fb_sdoread_6041(sNetId:= fb_netid, nSlaveAddr:=fb_nslaveaddr , nSubIndex:=0 , nIndex:=16#6041 , pDstBuf:=ADR(statusword) , cbBufLen:=2 , bExecute:=sdo_read , tTimeout:= , bBusy=> , bError=> , nErrId=> );
fb_sdoread_6060(sNetId:= fb_netid, nSlaveAddr:= fb_nslaveaddr, nSubIndex:=0 , nIndex:=16#6060 , pDstBuf:=ADR(mode_display) , cbBufLen:=1 , bExecute:=sdo_read , tTimeout:= , bBusy=> , bError=> , nErrId=> );
//fb_sdowrite_6060(sNetId:= fb_netid, nSlaveAddr:=fb_nslaveaddr , nSubIndex:=0 , nIndex:= 16#6060, pSrcBuf:=ADR(mode) , cbBufLen:=1 , bExecute:= mode<>mode_display AND sdo_read, tTimeout:= , bBusy=> , bError=> , nErrId=> );
fb_sdoread_607C(sNetId:= fb_netid, nSlaveAddr:=fb_nslaveaddr , nSubIndex:=0 , nIndex:=16#607C , pDstBuf:= ADR(home_offset_display), cbBufLen:=4 , bExecute:=sdo_read , tTimeout:= , bBusy=> , bError=> , nErrId=> );
fb_sdowrite_607C(sNetId:=fb_netid , nSlaveAddr:=fb_nslaveaddr , nSubIndex:=0 , nIndex:=16#607C , pSrcBuf:=ADR(home_offset) , cbBufLen:=4 ,	bExecute:=home_offset<>home_offset_display AND sdo_read , tTimeout:= , bBusy=> , bError=> , nErrId=> );
fb_sdoread_6098(sNetId:=fb_netid , nSlaveAddr:=fb_nslaveaddr , nSubIndex:=0 , nIndex:=16#6098 , pDstBuf:=ADR(home_method_display) , cbBufLen:=1 , bExecute:=sdo_read , tTimeout:= , bBusy=> , bError=> , nErrId=> );
fb_sdowrite_6098(sNetId:=fb_netid , nSlaveAddr:=fb_nslaveaddr , nSubIndex:=0 , nIndex:=16#6098 , pSrcBuf:=ADR(home_method) , cbBufLen:=1 , bExecute:=home_method<>home_method_display AND sdo_read , tTimeout:= , bBusy=> , bError=> , nErrId=> );
fb_sdoread_6099_01(sNetId:=fb_netid , nSlaveAddr:=fb_nslaveaddr , nSubIndex:=1 , nIndex:=16#6099, pDstBuf:=ADR(home_highspeed_display) , cbBufLen:=4 , bExecute:=sdo_read , tTimeout:= , bBusy=> , bError=> , nErrId=> );
fb_sdowrite_6099_01(sNetId:=fb_netid , nSlaveAddr:=fb_nslaveaddr , nSubIndex:=1 , nIndex:=16#6099 , pSrcBuf:=ADR(home_highspeed) , cbBufLen:=4 , bExecute:=home_highspeed<>home_highspeed_display AND sdo_read , tTimeout:= , bBusy=> , bError=> , nErrId=> );
fb_sdoread_6099_02(sNetId:=fb_netid , nSlaveAddr:=fb_nslaveaddr , nSubIndex:=2 , nIndex:=16#6099, pDstBuf:= ADR(home_lowspeed_display), cbBufLen:= 4, bExecute:=sdo_read , tTimeout:= , bBusy=> , bError=> , nErrId=> );
fb_sdowrite_6099_02(sNetId:=fb_netid , nSlaveAddr:=fb_nslaveaddr , nSubIndex:=2 , nIndex:=16#6099 , pSrcBuf:=ADR(home_lowspeed) , cbBufLen:=4 , bExecute:=home_lowspeed<>home_lowspeed_display AND sdo_read , tTimeout:= , bBusy=> , bError=> , nErrId=> );
fb_sdoread_6091_01(sNetId:=fb_netid , nSlaveAddr:=fb_nslaveaddr , nSubIndex:=1 , nIndex:=16#6091 , pDstBuf:= ADR(motor), cbBufLen:= 4, bExecute:=sdo_read , tTimeout:= , bBusy=> , bError=> , nErrId=> );
fb_sdoread_6091_02(sNetId:=fb_netid , nSlaveAddr:=fb_nslaveaddr , nSubIndex:=2 , nIndex:=16#6091 , pDstBuf:=ADR(shaft), cbBufLen:=4 , bExecute:=sdo_read , tTimeout:= , bBusy=> , bError=> , nErrId=> );
//fb_sdoread_6064(sNetId:=fb_netid , nSlaveAddr:=fb_nslaveaddr , nSubIndex:=2 , nIndex:=16#6099 , pSrcBuf:=ADR(home_lowspeed) , cbBufLen:=4 , bExecute:=home_lowspeed<>home_lowspeed_display AND sdo_read , tTimeout:= , bBusy=> , bError=> , nErrId=> );

IF iMode = 3 OR iMode =1 //雷赛伺服
THEN 
	mcsetposition(
		Axis:= axis_name, 
		Execute:= (statusword.10=TRUE AND  statusword.12=TRUE AND statusword.13=FALSE AND home_start), 
		Position:= 0, 
		Mode:= , 
		Options:= , 
		Done=> , 
		Busy=> , 
		Error=> , 
		ErrorID=> );
END_IF

IF home_exe THEN
home_start:=TRUE;
home_done := FALSE;//增加
//ELSE home_error:=TRUE; error_id:=8001; home_start:=FALSE;
END_IF

IF home_start (*AND FALSE*) THEN
	CASE home_step OF
		0://复位关闭
		exe_reset:=FALSE;	
		IF NOT(home_error) THEN
			home_step:=3;
			mcsetposition(
				Axis:= axis_name, 
				Execute:= FALSE);
		END_IF
		1://检测是否是三菱驱动器
		IF 	iMode = 1
		THEN 
			mcsetposition(
			Axis:= axis_name, 
			Execute:= TRUE, 
			Position:= 0, 
			Mode:= , 
			Options:= , 
			Done=> , 
			Busy=> , 
			Error=> , 
			ErrorID=> ); 
			IF mcsetposition.Done
			THEN
				mcsetposition(
					Axis:= axis_name, 
					Execute:= FALSE);
				home_step := 3;
			END_IF			
		ELSE
			home_step := 3; 
		END_IF
		
		3://将模式切为回原点模式6
		mode:=6;
		home_done := FALSE;
		ton2.IN:=TRUE;
		IF ton2.Q THEN
			ton2.IN:=FALSE;
			home_step:=5;
		END_IF
		5://将控制字改为F，上使能
        IF NOT home_error THEN
			controlword:=15;
			home_step:=10;
			ton2.IN:=FALSE;
		ELSE
			home_error:=TRUE;
			error_id:=8002;
			home_step:=0;
		END_IF
		10://复位
		exe_reset:=TRUE;
		ton2.IN:=TRUE;
		IF ton2.Q THEN 
			ton2.IN:=FALSE;
			home_step:=15;
		END_IF
		15://复位完成，控制字改为F
		IF reset_done AND statusword.1 THEN
			exe_reset:=FALSE;
			home_step:=25;
		ELSE
			home_error:=TRUE;
			error_id:=8003;
			home_step:=0;
		END_IF
		
		25://确认模式切换为6,与设定值相同
		IF mode=mode_display AND home_offset=home_offset_display AND home_method=home_method_display AND home_highspeed=home_highspeed_display AND home_lowspeed=home_lowspeed_display 
        AND (mode_display<>0) AND (home_method_display<>0) AND (home_highspeed_display<>0) AND (home_lowspeed_display<>0) AND (numerator<>0) AND (denominator<>0) THEN 
			home_step:=26;
			_tonDelay1(in:=FALSE);
			_tonDelay2(in:=FALSE);
		ELSE
			home_error:=TRUE;
			error_id:=8004;
			home_step:=0;
		END_IF
		
		26:
			controlword:=31;
			_tonDelay1(in:=TRUE,PT:=T#2S);
			IF _tonDelay1.Q THEN
				_tonDelay1(in:=FALSE);
				home_step:=30;
			END_IF		
		30://将控制字切为1F，启动回原点功能
		IF statusword.10 AND  statusword.12 AND NOT statusword.13 THEN
			home_step:=40;
		(*ELSIF statusword.13 THEN
			home_error:=TRUE;
			error_id:=8005;
			home_step:=0;	*)		
		ELSE
			_tonDelay2(IN:=TRUE,pt:=tTimeOutSet);
		END_IF
		
		(*_tonDelay1(in:=(statusword.10=TRUE) AND  statusword.12=TRUE AND statusword.13=FALSE,pt:=T#200MS);//回原点已经完成
		_tonDelay2(in:=( statusword.10=FALSE AND  statusword.12=FALSE AND statusword.13=TRUE ) OR ( statusword.10=FALSE AND  statusword.12=TRUE AND statusword.13=FALSE ) OR 
                       ( statusword.10=TRUE AND  statusword.12=FALSE AND statusword.13=FALSE ) OR ( statusword.10=TRUE AND  statusword.12=FALSE AND statusword.13=TRUE ) OR 
					   ( statusword.12=TRUE AND statusword.13=TRUE )	,pt:=T#10S);//会员店内失败
		IF _tonDelay1.Q  THEN//检测状态字回原点完成
			_tonDelay1(IN:=FALSE);
			home_step:=40;
		END_IF*)
		IF _tonDelay2.Q THEN
			_tonDelay2(IN:=FALSE);
			home_error:=TRUE;
			error_id:=8005;
			home_step:=0;
		END_IF
		40://复位
		//exe_reset:=TRUE;
		_tonDelay2(IN:=FALSE);
		ton2.IN:=(TRUE);
		IF ton2.Q THEN
			ton2.IN:=(FALSE);
			_tonDelay(IN:=FALSE);
			home_step:=41;
		END_IF
		41://增加断使能功能
		controlword:=0;
		_tonDelay(IN:=NOT statusword.1 , PT:=T#100MS , Q=> , ET=> );
		IF _tonDelay.Q THEN
			_tonDelay(IN:=FALSE);
			home_step:=45;
		END_IF

		45://将模式切换为位置模式8
//		IF reset_done THEN			
//			exe_reset:=FALSE;
//			_tonDelay(IN:=FALSE);
			home_step:=46;
//		ELSE
//			home_error:=TRUE;
//			error_id:=8006;
//			home_step:=0;
//		END_IF
		46://增加上使能功能
		//controlword:=15;
		_tonDelay(IN:=TRUE , PT:=T#1S , Q=> , ET=> );
		IF _tonDelay.Q THEN
			_tonDelay(IN:=FALSE);
			home_step:=50;
		END_IF		
		50:
		_iCount := _iCount + 1 ;
		mode:=8;
		home_done:=TRUE;
		exe_reset:=FALSE;
		home_start:=FALSE;
		home_step:=0;
	END_CASE
END_IF


(*IF NOT(home_exe)THEN
	home_step:=0;
	home_error:=FALSE;
	home_done:=FALSE;
	home_start:=FALSE;
	error_id:=0;
END_IF*)

IF home_error THEN
	home_step:=0;
	//
	home_done:=FALSE;
	home_start:=FALSE;
	exe_reset:=TRUE;
	IF reset_done THEN
		error_id:=0;
		mode:=8;
		home_error:=FALSE;
		exe_reset:=FALSE;
	END_IF
END_IF

END_FUNCTION_BLOCK

// ---- POUs/003_FB/17_HMIFB/FB_Proface.TcPOU
FUNCTION_BLOCK FB_Proface
VAR_INPUT
	xEStop								: BOOL;					//急停
	xSafety								: BOOL;					//安全防护
	xManualMode							: BOOL;					//手动模式
	xAutoMode							: BOOL;					//自动模式
	xAlarm								: BOOL;					//报警中
	xTip								: BOOL;					//提示中
	xInit								: BOOL;					//初始化
	xIniting							: BOOL;					//初始化中
	xInitDone							: BOOL;					//初始化完成
	xDummyChecking						: BOOL;					//点检中
	xDummyCheckDone						: BOOL;					//点检完成
	xEmptying							: BOOL;					//清料中
	xEmptyDone							: BOOL;					//清料完成
	xStartHmi							: BOOL;					//启动HMI
	xStopHmi							: BOOL;					//停止HMI
	xResetHmi							: BOOL;					//复位HMI
	xPauseHmi							: BOOL;					//暂停HMI
	xInitHmi							: BOOL;					//初始化HMI
	xInitConfirmHmi						:BOOL;					//测试使用
	xManualModeHmi						: BOOL;					//手动HMI
	xAutoModeHmi						: BOOL;					//自动HMI
	xUnlockHmi							: BOOL;					//解锁HMI
	xDummyCheckHmi						: BOOL;					//点检HMI
	xEmptyHmi							: BOOL;					//清料HMI
	xWindowColseHmi						: BOOL;					//窗口关闭HMI
	                      		
	nCurrentPageIndex					: UINT:=0;				//当前画面索引
	nJumpToPageIndex					: UINT:=1;				//跳转到画面索引
	                      		
	nWindowControlIndex					: UINT:=0;				//窗口控制索引
	nWindowNumberIndex					: UINT:=1;				//窗口编号索引
	nWindowLocationIndexX				: UINT:=2;				//窗口位置索引X坐标
	nWindowLocationIndexY				: UINT:=3;				//窗口位置索引Y坐标
	                      		
	nWindowLocationX					: UINT:=300;			//窗口位置X坐标
	nWindowLocationY					: UINT:=80;		    //窗口位置Y坐标
	                      		
	nInitConfirmWindow					: UINT:=1;				//初始化确认窗口编号
	nInitAlarmWindow					: UINT:=2;				//初始化有报警窗口编号
	nInitingAlarmWindow					: UINT:=3;				//初始化中有报警窗口编号
	nInitingWindow						: UINT:=4;				//初始化中窗口编号
	nInitDoneWindow						: UINT:=5;				//初始化完成窗口编号
	nInitFailWindow						: UINT:=6;				//初始化失败窗口编号
	
	nDummyCheckConfirmWindow			: UINT:=5;				//点检确认窗口编号
	nDummyCheckDoneWindow				: UINT:=6;				//点检完成窗口编号
	nDummyCheckFailWindow				: UINT:=7;				//点检失败窗口编号
	
	nEmptyConfirmWindow					: UINT:=10;				//清料确认窗口编号
	nEmptyDoneWindow					: UINT:=11;				//清料完成窗口编号
	
	nTipWindow							: UINT:=31;				//提示窗口编号
	nButtonWindow						: UINT:=121;			//调试窗口编号
END_VAR

VAR_OUTPUT
END_VAR

VAR
	
	xStartLight							: BOOL;					//启动灯
	xStopLight							: BOOL;					//停止灯
	xResetLight							: BOOL;					//复位灯
	xPauseLight							: BOOL;					//暂停灯
	xInitLight							: BOOL;					//初始化灯
	
END_VAR

VAR
	
	wSystem								: ARRAY[0..20] OF WORD;	//系统区
	wWindow								: ARRAY[0..20] OF WORD;	//窗口控制区
	                  				
	ftTip								: F_TRIG;				//提示中下降沿
	rtInit								: R_TRIG;				//初始化上升沿
	ftIniting							: F_TRIG;				//初始化中下降沿
	rtDummyCheck						: R_TRIG;				//点检上升沿
	ftDummyChecking						: F_TRIG;				//点检中下降沿
	rtEmptyConfirm						: R_TRIG;				//清料确认上升沿
	rtEmptyDone							: R_TRIG;				//清料完成上升沿
	
END_VAR

ACT_Init();
ACT_DummyCheck();
ACT_Empty();
ACT_Control();

ACTION ACT_Control:
ftTip(CLK:=xTip, Q=>);
IF xWindowColseHMI		//窗口关闭
	OR ftTip.Q			//提示下降沿自动关闭窗口
THEN
	wWindow[nWindowNumberIndex]:=0;
END_IF

//IF xTip THEN
//	wWindow[nWindowNumberIndex]:=nTipWindow;
//END_IF

wWindow[nWindowControlIndex].0:=wWindow[nWindowNumberIndex]<>0;

wWindow[nWindowLocationIndexX]:=nWindowLocationX;
wWindow[nWindowLocationIndexY]:=nWindowLocationY;
END_ACTION

ACTION ACT_DummyCheck:
rtDummyCheck(CLK:=xDummyCheckHmi, Q=>);
ftDummyChecking(CLK:=xDummyChecking, Q=>);
IF rtDummyCheck.Q	//点检确认窗口显示
	AND xEStop
	AND xSafety
	AND xManualMode
	AND xInitDone
	AND NOT xAlarm
THEN
	wWindow[nWindowNumberIndex]:=nDummyCheckConfirmWindow;
END_IF
IF ftDummyChecking.Q THEN
	IF xDummyCheckDone THEN		//点检完成窗口显示
		wWindow[nWindowNumberIndex]:=nDummyCheckDoneWindow;
	ELSE	//点检失败窗口显示
		wWindow[nWindowNumberIndex]:=nDummyCheckFailWindow;
	END_IF
END_IF
END_ACTION

ACTION ACT_Empty:
rtEmptyConfirm(CLK:=xEmptyHmi, Q=>);
rtEmptyDone(CLK:=xEmptyDone, Q=>);
IF rtEmptyConfirm.Q		//清料确认窗口显示
	AND fbMachine[1].xEStop
	AND fbMachine[1].xSafety
	AND fbMachine[1].xAutoMode
	AND fbMachine[1].xInitDone
	AND NOT fbMachine[1].xAlarm
THEN
	wWindow[nWindowNumberIndex]:=nEmptyConfirmWindow;
END_IF

IF rtEmptyDone.Q THEN	//清料完成窗口显示
	wWindow[nWindowNumberIndex]:=nEmptyDoneWindow;
END_IF
END_ACTION

ACTION ACT_Init:
rtInit(CLK:=xInit, Q=>);
ftIniting(CLK:=xIniting, Q=>);

IF rtInit.Q
THEN
	wSystem[0]:=10;
END_IF

IF rtInit.Q					//初始化确认窗口显示
	AND xEStop
	AND xSafety
	AND xManualMode
	AND NOT xAlarm
	AND NOT xIniting
THEN
	wWindow[nWindowNumberIndex]:=nInitConfirmWindow;
END_IF

IF rtInit.Q					//初始化有报警
	AND xAlarm
THEN
	wWindow[nWindowNumberIndex]:=nInitAlarmWindow;
END_IF

IF xIniting					//初始化中有报警
	AND xAlarm
THEN
	wWindow[nWindowNumberIndex]:=nInitingAlarmWindow;
END_IF

IF xIniting THEN			//初始化中窗口显示
	wWindow[nWindowNumberIndex]:=nInitingWindow;
END_IF

IF ftIniting.Q THEN		
	IF xInitDone THEN		//初始化完成窗口显示
		wWindow[nWindowNumberIndex]:=nInitDoneWindow;
	ELSE					//初始化失败窗口显示
		wWindow[nWindowNumberIndex]:=nInitFailWindow;
	END_IF
END_IF

IF xWindowColseHMI
THEN
	wWindow[nWindowNumberIndex]:=0;
	wWindow[nWindowControlIndex]:=0;
END_IF
END_ACTION

END_FUNCTION_BLOCK

// ---- POUs/003_FB/14_MachineFB/FB_Machine.TcPOU
FUNCTION_BLOCK  FB_Machine
VAR_INPUT
	xEStop						: BOOL;					//急停(运行时常ON)
	xKey						: BOOL;					//钥匙开关
	xDoorClosed					: BOOL;					//所有安全门关好
	xSafety						: BOOL;					//安全防护中
	xAirOn						: BOOL;					//气压正常
	xAlarm						: BOOL;					//报警中
	xManualTip					: BOOL;					//手动提示中
	xAutoTip					: BOOL;					//自动提示中
	xTip						: BOOL;					//提示中
	
	xStart						: BOOL;					//启动按钮
	xStop						: BOOL;					//停止按钮
	xReset						: BOOL;					//复位按钮
	xPause						: BOOL;					//暂停按钮
	xInit						: BOOL;					//初始化按钮
	xManualMode					: BOOL;					//手动模式
	xAutoMode					: BOOL;					//自动模式

	
	xInitConfirm				: BOOL;					//初始化确认
	xInitDone					: BOOL;					//初始化完成
	tInitTimeout				: TIME:=T#3M;			//初始化超时延时
	
	xDummyMode					: BOOL;					//点检模式，点检使能
	xStationDummyDone			: BOOL;					//工站点检完成
	xDummyDone					: BOOL;					//点检完成
	xDummyDoneConfirm			: BOOL;					//点检完成确认
	
	xSampling					: BOOL;					//取样中
	uiSampleCount				: UINT;					//取样数量统计
	xSampleDone					: BOOL;					//取样完成
	xEmptyHmi					: BOOL;					//清料HMI
	xEmptyConfirmHmi			: BOOL;					//清料确认HMI
	xEmptyDone					: BOOL;					//清料完成
	xOrderFinished				: BOOL;					//订单完成
	xOrderChanged				: BOOL;					//订单切换
	
	xTryRun						: BOOL;					//空跑试运行
	xCycleEnable      	 		: BOOL;          		//设备CT计时
	xDataEmpty					: BOOL;					//数据清空
	tDataEmpty					: TIME;					//数据清空延时，默认为0
	xCarrierDataClear			: BOOL;					//载座数据清空
	tCarrierDataClear			: TIME;					//载座数据清空延时，默认为0
	
	xInitConfirmDialog			: BOOL;					//初始化确认对话框
	
	dwStatus					:ARRAY[1..4] OF DWORD;	//状态，bit.0急停中.1钥匙关闭.2气压低.3手动模式.4自动模式.5未准备好.6准备就绪.7运行中.8停止中.9报警中.10暂停中.11初始化中.12清料中.13清料完成.14取样中.15取样完成.16订单完成.17点检屏蔽中.18要求点检.其它可自定义	
 
	dwMessage					:ARRAY[1..5] OF DWORD;	//提示信息
	dwAlarm						:ARRAY[1..5] OF DWORD;	//报警信息	
	
	xDummyDisabled				: REFERENCE TO BOOL;	//点检屏
	//rCycleTime				: REAL;					//生产周期，单位s
	//生产信息相关变量
	xClearCountData 			: BOOL ; //清除产量数据
	udiGoods					: UDINT;				//当前良品数量
	udiBads						: UDINT;				//当前不良数量
	udiTotal					:  UDINT;				//当前总数量
	rYield						:  REAL;				//当前良品率
	rReject						:  REAL;				//当前不良率
END_VAR

VAR_OUTPUT
	xEStopped					: BOOL;					//急停状态
	xRunning					: BOOL;					//自动中
	xStopped					: BOOL;					//停止状态
	xPaused						: BOOL;					//暂停状态
	xIniting					: BOOL;					//初始化中
	xEmptying					: BOOL;					//清料中
	
	xAutoModeTip				: BOOL;					//自动模式上升沿提示
	
	xInitTimeout				: BOOL;					//初始化超时
	xReInit						: BOOL;					//整机重新初始化，用于复位各工站初始化完成
	
	xInitDoneDialog				: BOOL;					//初始化完成对话框
	xInitFailedDialog			: BOOL;					//初始化失败对话框
	
	xEmptyConfirmDialog			: BOOL;					//清料确认对话框
	xEmptyDoneDialog			: BOOL;					//清料完成对话框
	
	xShowAlarm					: BOOL;					//报警信息显示
	xShowTip					: BOOL;					//提示信息显示
	
	xStartLight					: BOOL;					//启动按钮灯
	xStopLight					: BOOL;					//停止按钮灯
	xResetLight					: BOOL;					//复位按钮灯
	xPauseLight					: BOOL;					//暂停按钮灯
	xInitLight					: BOOL;					//初始化按钮灯
	
	xLampGreen					: BOOL;					//三色灯-绿
	xLampYellow					: BOOL;					//三色灯-黄
	xLampRed					: BOOL;					//三色灯-红
	xLampBuzzer					: BOOL;					//三色灯-蜂鸣器	
	
	diLastCycleTime				:DINT;					//基础时间是100ms
	diCycleTime        			: DINT;					//基础时间是100ms

END_VAR

VAR
	{attribute 'hide'}
	rtRunning					: R_TRIG;				//自动中上升沿
	{attribute 'hide'}
	rtEmptyDone					: R_TRIG;				//清料完成上升沿
	{attribute 'hide'}
	tonDataEmpty				: TON;					//数据清零延时
	rtDataEmpty					: R_TRIG;				//数据清空上升沿
	{attribute 'hide'}
	tonCarrierDataClear			: TON;					//载座数据清空延时
	rtCarrierDataClear			: R_TRIG;				//载座数据清空上升沿
	{attribute 'hide'}
	xDummyWarnTime				: BOOL;					//点检提醒时间
	{attribute 'hide'}
	rtDummyWarnTime				: R_TRIG;				//点检提醒时间上升沿
	{attribute 'hide'}
	xDummyAlarmTime				: BOOL;					//点检报警时间
	{attribute 'hide'}
	rtDummyAlarmTime			: R_TRIG;				//点检报警时间上升沿
	{attribute 'hide'}
	rtDummyDoneConfirm			: R_TRIG;				//点检完成确认上升沿
	{attribute 'hide'}
	xDummyDoneCache				: BOOL;					//点检完成缓存
	{attribute 'hide'}
	xDummyComplete				: BOOL;					//点检完成状态
	{attribute 'hide'}
	xDummyRequirement			: BOOL;					//要求点检提醒
	{attribute 'hide'}
	rtInit						: R_TRIG;				//初始化上升沿
	{attribute 'hide'}
	rtInitConfirm				: R_TRIG;				//初始化确认上升沿
	{attribute 'hide'}
	ftIniting					: F_TRIG;				//初始化下降沿
	{attribute 'hide'}
	rtEmptyHmi					: R_TRIG;				//清料HMI上升沿
	{attribute 'hide'}
	ftEmptying					: F_TRIG;				//清料中下降沿
	{attribute 'hide'}
	xInitAble					: BOOL;					//初始化条件
	{attribute 'hide'}
	xRunAble					: BOOL;					//运行条件
	{attribute 'hide'}
	tonInitTimeout				: TON;					//初始化超时
	{attribute 'hide'}
	tonLampBuzzer				: TON;					//蜂鸣器关闭延时
	{attribute 'hide'}
	rtCycleFlag					: R_TRIG;				//循环标志上升沿
	{attribute 'hide'}
	lrCycleTimer				: LREAL;				//计时器，单位100ns，除于10000后单位ms
	{attribute 'hide'}
	tonHydraGoodsOut			: TON;					//Hydra良品输出信号延时
	{attribute 'hide'}
	tonHydraGoodsInterval		: TON;					//Hydra良品输出信号间隔
	{attribute 'hide'}
	tonHydraBadsOut				: TON;					//Hydra不良输出信号延时
	{attribute 'hide'}
	tonHydraBadsInterval		: TON;					//Hydra不良输出信号间隔
	
	rtAutoMode					: R_TRIG;				//自动模式上升沿
	rMachineStart       		: R_TRIG;
	i : INT ;

END_VAR

ACT_General();
ACT_Init();
ACT_Empty();
ACT_Start();
ACT_Pause();
ACT_Stop();
ACT_Reset();
ACT_Lamp();
ACT_Data();
ACT_CycleTime();

ACTION ACT_CycleTime:
//	初始化时同时初始化工站周期计时
IF xIniting THEN
	xCycleEnable:=FALSE;
END_IF

//工站完成触发信号
rMachineStart(CLK:= xCycleEnable);
IF rMachineStart.Q
THEN
	diCycleTime:=diLastCycleTime;
	diLastCycleTime := 0;
END_IF
//	工站周期计时
IF xRunning AND xCycleEnable AND stSysPulse.xR100ms
THEN
	diLastCycleTime := diLastCycleTime + 1;//对应最小周期是0.1ms
END_IF
END_ACTION

ACTION ACT_Data:
//	当前数据清零
tonDataEmpty(IN:=xDataEmpty, PT:=tDataEmpty, Q=> , ET=> );
rtDataEmpty(CLK:=tonDataEmpty.Q, Q=> );
IF rtDataEmpty.Q THEN
	udiGoods:=0;
	udiBads:=0;
END_IF

//	计算当前良品率
udiTotal:=udiGoods + udiBads;
IF udiTotal > 0 THEN
	rYield:=LREAL_TO_REAL(100 * UDINT_TO_LREAL(udiGoods) / UDINT_TO_LREAL(udiTotal));
	rReject:=100.0 - rYield;
ELSE
	rReject:=0;
	rYield:=0;
END_IF



//	转台数据清零上升沿
tonCarrierDataClear(IN:=xCarrierDataClear, PT:=tCarrierDataClear, Q=> , ET=> );
rtCarrierDataClear(CLK:=tonCarrierDataClear.Q, Q=> );
END_ACTION

ACTION ACT_Empty:
//	启动时，先复位清料完成
IF xStart
	AND NOT xRunning
	AND NOT xEmptying
THEN
	xEmptyDone:=FALSE;
END_IF

//	清料HMI上升沿，弹出清料确认对话框
rtEmptyHmi(CLK:=xEmptyHmi, Q=> );
xEmptyConfirmDialog:=rtEmptyHmi.Q
	AND xEStop
	AND xKey
	AND xSafety
	AND xInitDone
	AND NOT xAlarm
	AND NOT xTip
	AND NOT xIniting;

//	清料
IF xEStop
	AND NOT xIniting
	AND NOT xEmptyDone
THEN
	IF xEmptyConfirmHmi
		AND xKey
		AND xSafety
		AND xInitDone
		AND NOT xAlarm
		AND NOT xTip
	THEN
		xEmptying:=TRUE;
		xEmptyConfirmHmi := FALSE ;
	END_IF
ELSE
	xEmptying:=FALSE;
END_IF

//	清料中下降沿，弹出清料完成对话框
ftEmptying(CLK:=xEmptying, Q=> );
xEmptyDoneDialog:=ftEmptying.Q
	AND xEmptyDone;
END_ACTION

ACTION ACT_General:
//	急停中
xEStopped:=NOT xEStop;

xShowAlarm := FALSE;
FOR i:=1 TO 4 BY 1 DO 	
 IF dwMessage[i]<>0 THEN 
		xShowAlarm := TRUE ;
		EXIT ;
 END_IF
END_FOR
//提示报警显示
xShowAlarm:= xShowAlarm OR xAlarm;

//提示信息显示
xShowTip:=xTip;

//报警复位
IF xReset THEN
	FOR i:=1 TO 5 BY 1 DO 
		dwMessage[i] := dwAlarm[i]  := 0;
	END_FOR
END_IF
END_ACTION

ACTION ACT_Init:
//	初始化条件
xInitAble:=xEStop
	AND xKey
	AND xSafety
	AND xManualMode
	AND NOT xAlarm
	AND NOT xInitTimeout;

//	初始化上升沿，弹出初始化确认对话框
rtInit(CLK:=xInit, Q=> );
IF rtInit.Q AND xInitAble AND NOT xIniting THEN
  xInitConfirmDialog :=TRUE;	
END_IF
(*bInitConfirmDialog:=rtInit.Q
	AND bInitAble
	AND NOT bIniting;*)

//	初始化确认上升沿，触发各工站重新初始化
rtInitConfirm(CLK:=xInitConfirm, Q=> );
xReInit:=rtInitConfirm.Q
	AND xInitAble
	AND NOT xIniting;
//false初始化弹出的窗口
IF rtInitConfirm.Q
THEN 
  xInitConfirmDialog :=FALSE;
  
END_IF

//	初始化中
IF xInitAble
	AND NOT xPause
	AND NOT xInitDone
THEN
	IF xInitConfirm THEN
		xIniting:=TRUE;
	END_IF
ELSE
	xIniting:=FALSE;
END_IF

//	初始化按钮灯，初始化中闪烁，初始化完成熄灭
xInitLight:=xIniting AND stSysPulse.xP1s ;

//	初始化超时
tonInitTimeout(
	IN:=xIniting,
	PT:=tInitTimeout,
	Q=> , ET=>
);
IF xReset THEN
	xInitTimeout:=FALSE;
END_IF
IF tonInitTimeout.Q THEN
	xInitTimeout:=TRUE;
END_IF

//	初始化中下降沿，弹出初始化完成或失败对话框
ftIniting(CLK:=xIniting, Q=> );
xInitDoneDialog:=ftIniting.Q
	AND xInitDone;
xInitFailedDialog:=ftIniting.Q
	AND NOT xInitDone;
END_ACTION

ACTION ACT_Lamp:
//	三色灯-绿，运行中绿灯常亮
xLampGreen:=xRunning OR xStartLight;

//	三色灯-红，报警或急停中红灯常亮
xLampRed:=xAlarm OR xEStopped;

//	三色灯-黄，其余情况下黄灯常亮，有等待信息时黄灯闪烁

xLampYellow:=NOT xLampGreen AND NOT xLampRed AND  (stSysPulse.xP1s OR (xinitdone AND xmanualmode));	




//	蜂鸣器关闭延时
tonLampBuzzer(IN:=xAlarm, PT:=T#3S, Q=> , ET=> );

//	三色灯-蜂鸣器
xLampBuzzer:=xAlarm
	AND stSysPulse.xP1s
	AND NOT tonLampBuzzer.Q;
END_ACTION

ACTION ACT_Pause:
//	暂停中
IF xPause  THEN
	xPaused:=TRUE;
END_IF

IF xEStopped
	OR xStart
THEN
	xPaused:=FALSE;
END_IF

//暂停按钮灯，暂停中常亮
xPauseLight:=xPaused;
END_ACTION

ACTION ACT_Reset:
//	复位按钮灯，报警时闪烁
xResetLight:=xAlarm
	AND stSysPulse.xP1s;
END_ACTION

ACTION ACT_Start:
//	运行条件
xRunAble:=xEStop
	AND xKey
	AND xSafety
	AND xAutoMode
	AND xInitDone
	AND NOT xAlarm
	AND NOT xAutoTip
	AND NOT xStopped;

//	运行中
IF xRunAble
	AND NOT xPause
	AND NOT xEmptyDone//清料完成
THEN
	IF xStart THEN
		xRunning:=TRUE;
	END_IF
ELSE
	xRunning:=FALSE;
END_IF

//	启动按钮灯，运行中常亮，准备就绪时闪烁
xStartLight:=xRunning
	OR xRunAble
		AND stSysPulse.xP1s;
END_ACTION

ACTION ACT_Stop:
//	停止中
IF xStop AND xRunning THEN
	xStopped:=TRUE;
END_IF

IF xEStopped
	OR xStart
	OR xPaused
THEN
	xStopped:=FALSE;
END_IF

//停止按钮灯，停止中常亮
xStopLight:=xStopped;
END_ACTION

END_FUNCTION_BLOCK

// ---- POUs/003_FB/53_RudongPump/08_PeristalticPumpFB/FB_RuDongPump_modbus_DF600Plus.TcPOU
//{attribute 'tc_no_symbol'}
FUNCTION_BLOCK FB_RuDongPump_modbus_DF600Plus
VAR_INPUT
	xExecute: BOOL;
	xAbort: BOOL;
	xResetRequest: BOOL;//匹配复位按钮 
	xRunILC		:BOOL:=TRUE;//蠕动泵运行条件
	dwTimeLimit: DWORD:=1;//[ms],1 => no invocation time limit
	dwTimeOut: DWORD;//[ms],0 => no executing time limit
	stPara       : RudongPump_Sys_Para;				
	xNeedConfigurePara		: BOOL := TRUE;//是否需要配置参数(默认是需要进行参数配置的)	
	stRunPara	:RudongPump_RunData;//运行参数	
	xAutoMode    : BOOL;//0:mannal 1:auto
	xIniting     : BOOL;//初始化过程中
	xDeviceRunning : BOOL;//工站单循环中
	rSpeedRatio  : REAL:=2.733;//根据泵头软管型号不同有变化
	sHmiError : STRING;
	xEStop : BOOL;
	stDeviceOpe	: RudongPump_Ope;//操作按钮
	stModbusAddress:ST_ModbusAddress;
	iDirectionSet:INT;
END_VAR
VAR_OUTPUT
	xDone: BOOL;(*完成条件满足*)
	xBusy: BOOL;(*动作正在执行*)
	xError	:BOOL;//报警中
	xAborted: BOOL;(*指令被打断*)
	xRunning	:BOOL;//蠕动泵运行中
	xRudongPump_ERROR: BOOL;(*错误条件满足*)
	eERRORID: RudongPump_ERROR;(*错误码*)
	eMobbusErrorID : UDINT;//modubs 报警信息
	xRdyCmd : BOOL;
	iMaxRunTime	:REAL;//最大运行时间,单位s
	iMinRunTime	:REAL;//最小运行时间,单位s
END_VAR
VAR_IN_OUT
		
END_VAR
VAR
{attribute 'tc_no_symbol'}
	eState: STATE;
{attribute 'tc_no_symbol'}
	_xDone: BOOL;
{attribute 'tc_no_symbol'}
	eCmd : RudongPump_CMD;//指令控制	
{attribute 'tc_no_symbol'}
	xFirstInvocation: BOOL := TRUE;	
{attribute 'tc_no_symbol'} 
	xTimeOut: BOOL;
{attribute 'tc_no_symbol'}
	xTimeLimit: BOOL;
{attribute 'tc_no_symbol'}
	tInvocationTimer , tOperationTimer : TON;
{attribute 'tc_no_symbol'}
	rFluVolumeSet   : REAL;//液量设定 0.0-99999.0 mL(0.1ml)
{attribute 'tc_no_symbol'}
	rRuntimeSet     : REAL;//运行时间设定 0.1-9999s(0.1s)
{attribute 'tc_no_symbol'}
	iCycleNumber		: INT;//重复次数
{attribute 'tc_no_symbol'}
	iModuleAdress		: INT;//灌装单元地址
{attribute 'tc_no_symbol'}
	iModuleSpeed		: REAL;//灌装单元速度
{attribute 'tc_no_symbol'}
	iModuleRealVolume	: REAL;//灌装实际液量	
{attribute 'tc_no_symbol'}	
	iBackAngle	:INT;
{attribute 'tc_no_symbol'}
	_cmdStop  : BOOL;  
{attribute 'tc_no_symbol'}
	_tonTimeout , _tonCmdTimeout : TON;	
{attribute 'tc_no_symbol'}
  /// command execution
  _CmdExe : BOOL;
{attribute 'tc_no_symbol'}
  /// detect rising edge of command execution
  _rTrigCmdExe : R_TRIG;
{attribute 'tc_no_symbol'}	
  _rTrigCmdOrg   : R_TRIG;	
{attribute 'tc_no_symbol'}
	_diCmdState 	: DINT; 
{attribute 'tc_no_symbol'} 
  /// detect FltQuit rising edge
  _rTrigFltReset      : R_TRIG; 
{attribute 'tc_no_symbol'} 
  _tonDelay : TON; 
{attribute 'tc_no_symbol'}	
	_iConnectState : INT := 0;
{attribute 'tc_no_symbol'}	
	_connectTon : TON;
{attribute 'tc_no_symbol'}		
	_xConnectError : BOOL;
{attribute 'tc_no_symbol'}		
	_fResetCheck : F_TRIG;
{attribute 'tc_no_symbol'}		
	_rManual : R_TRIG;
{attribute 'tc_no_symbol'}		
	_fManual : F_TRIG;
{attribute 'tc_no_symbol'}		
	_xModeChange : BOOL;
{attribute 'tc_no_symbol'}		
	i : INT;
{attribute 'tc_no_symbol'}		
	_tonPulse : TON;//状态读取计时定时器
{attribute 'tc_no_symbol'}		
  _xCheckModbusRun : BOOL;//检测modbus是否处理总
{attribute 'tc_no_symbol'}	  
	_xConfigureParaOK : BOOL;//需要匹配参数是OK的
{attribute 'tc_no_symbol'}		
	_rStopCmdTrig : R_TRIG;
{attribute 'tc_no_symbol'}		
	_iActRunNumber : INT ;//当前运行的次数
{attribute 'tc_no_symbol'}		
	_wFluVolumeSetTemp : WORD;
{attribute 'tc_no_symbol'}		
	_wRuntimeSetTemp : WORD;
{attribute 'tc_no_symbol'}		
	_wSpeedSetTemp : WORD;	
{attribute 'tc_no_symbol'}		
	_rSetSpeed : REAL;
{attribute 'tc_no_symbol'}		
	_wModuleSpeedSetTemp:WORD;
{attribute 'tc_no_symbol'}		
	_wModuleRealVolumeTemp:WORD;
{attribute 'tc_no_symbol'}		
	_rHMIControl : R_TRIG;
{attribute 'tc_no_symbol'}		
	dwTest1 : DWORD ;
{attribute 'tc_no_symbol'}		
	_iNGCount : INT;//NG 计数
{attribute 'tc_no_symbol'}		
	_rOperaTrig	:ARRAY [1..15] OF R_TRIG;
{attribute 'tc_no_symbol'}		
	k : INT;
{attribute 'tc_no_symbol'}		
	_bChannelNum , _bDiagData : BYTE;
{attribute 'tc_no_symbol'}		
	xAutomodeFlag	:BOOL;
{attribute 'tc_no_symbol'}		
	diStepOld:DINT;
{attribute 'tc_no_symbol'}			
	st_IOData : RudongPump_IOData;
{attribute 'tc_no_symbol'}		
	iPumpType	:INT;
{attribute 'tc_no_symbol'}	
	_xHMIOpe :BOOL;//是否有手动操作，是否有自动操作	
{attribute 'tc_no_symbol'}	
	 _xAutoOpe : BOOL;//是否有手动操作，是否有自动操作	
{attribute 'tc_no_symbol'}	
	_rInit	:R_TRIG;
{attribute 'tc_no_symbol'}		
	_first:BOOL;
{attribute 'tc_no_symbol'}				
	_aWrite_VAR: FB_MBWriteRegs;
{attribute 'tc_no_symbol'}
	_aRead_VAR: FB_MBReadRegs;	  
{attribute 'tc_no_symbol'}
//1:泵头型号；2:软管型号；3:启停控制	4:方向控制  5:全速运行  6:设定液量  7:时间设定  8:运行模式  9:重复次数		
//10:灌装单元地址  11:灌装单元速度  12:灌装单元启停  13:实际灌装量  14:灌装液量微调  15:恢复校准系数 	
// 设备反馈---------16:设备运行  17:设备校准中			
  _aExecute : ARRAY[1..17] OF BOOL;    
{attribute 'tc_no_symbol'}	
  _aQuantity : ARRAY[1..17] OF WORD:=[1,1,1,1,1,2,2,1,1,1,2,1,2,1,1,1,1];  //寄存器个数   
{attribute 'tc_no_symbol'}	
  _aMBAddr : ARRAY[1..17] OF WORD:=[1000,1001,1011,1010,1012,1002,1004,1022,1008,2000,2001,2003,2004,2006,2007,1011,2003];  //起始地址    
{attribute 'tc_no_symbol'}	
  _aAddr : ARRAY[1..17,1..2] OF  INT;  //存放区域                                                                                     
{attribute 'tc_no_symbol'}	
	_rxState:INT;
{attribute 'tc_no_symbol'}	
	_tonDelay1:TON;
{attribute 'tc_no_symbol'}		
	_iComNGCount:INT;
{attribute 'tc_no_symbol'}			
	_xBusy:BOOL;
{attribute 'tc_no_symbol'}			
	_xError:BOOL;	
{attribute 'tc_no_symbol'}		
	_iChannelIndex:INT;
END_VAR
VAR_TEMP
{attribute 'tc_no_symbol'}	
	xAgain: BOOL;
END_VAR

xAgain:=0;
ConnectAction();//触发通信连接功能连接
ACTMap();//IO Map
//ACT_GetModbusAdr();
IF NOT _first THEN
	_first:=TRUE;
ELSE

//只有在运行的时候，才会检测是否有模式切换发生
IF eState <> STATE.DORMANT
THEN	
	IF _rManual.Q OR _fManual.Q
	THEN
		_xModeChange := TRUE;//通知系统有模式切换发生
	END_IF
ELSE
	_xModeChange := FALSE;//待机状态不触发模式切换
END_IF

//检测是否是初始化中，如果是的去切换模式
_rInit(CLK:= xIniting);
IF _rInit.Q
THEN
	eState := STATE.RESETING;
END_IF	

REPEAT
	CASE eState OF
		STATE.DORMANT:
				HandleDormantState(xAgain=> xAgain);
		STATE.EXECUTING:
				HandleExecutingState(xAgain=> xAgain);
		STATE.DONE:
				HandleDoneState(xAgain=> xAgain);
		STATE.INERROR:
				HandleErrorState(xAgain=> xAgain);
		STATE.ABORTING:
				HandleAbortingState(xAgain=> xAgain);
		STATE.ABORTED:
				HandleAbortedState(xAgain=> xAgain);
		STATE.RESETING:
				HandleResettingState(xAgain=> xAgain);
	END_CASE
UNTIL (xAgain=0)
END_REPEAT
END_IF


//判断是否处于当前流程的Done状态
xDone := _xDone AND xExecute;
//输出报错信息
CASE eERRORID OF 	
  RudongPump_ERROR.No_ERROR:
		sHmiError:='No_ERROR';	
  RudongPump_ERROR.FLT_PARA:
		sHmiError:='FLT_PARA';
  RudongPump_ERROR.FLT_CONNECT:
		sHmiError:='FLT_CONNECT';
  RudongPump_ERROR.FLT_RDYCMD:
		sHmiError:='FLT_RDYCMD';
	RudongPump_ERROR.FLT_CONFIGURE_PARA:
		sHmiError:='FLT_CONFIGURE_PARA';
	RudongPump_ERROR.FLT_FLUVOLUM_TIME_PARA:
		sHmiError:='FLT_FLUVOLUM_TIME_PARA';  
  RudongPump_ERROR.FLT_PUSH_TIMEOUT:
		sHmiError:='FLT_PUSH_TIMEOUT';
  RudongPump_ERROR.FLT_PULL_TIMEOUT:
		sHmiError:='FLT_PULL_TIMEOUT';
  RudongPump_ERROR.FLT_STOP_TIMEOUT:
		sHmiError:='FLT_STOP_TIMEOUT'; 
	RudongPump_ERROR.FLT_FULLSPEEDSTOP_TIMEOUT:
		sHmiError:='FLT_FULLSPEEDSTOP_TIMEOUT';
	RudongPump_ERROR.FLT_FULLSPEEDSTART_TIMEOUT:
		sHmiError:='FLT_FULLSPEEDSTART_TIMEOUT'; 
	RudongPump_ERROR.FLT_CMD_TIMEOUT:
		sHmiError:='FLT_CMD_TIMEOUT';
	RudongPump_ERROR.FLT_RUN_FALL:
		sHmiError:='FLT_RUN_FALL';
END_CASE
//手动自动操作检测
_xHMIOpe :=
			stDeviceOpe.xConfigure_Hmi OR 
			stDeviceOpe.xFullSpeedPull_Hmi OR 
			stDeviceOpe.xFullSpeedPush_Hmi OR 
			stDeviceOpe.xPull_Hmi[1] OR 
			stDeviceOpe.xPull_Hmi[2] OR 
			stDeviceOpe.xPull_Hmi[3] OR 
			stDeviceOpe.xPull_Hmi[4] OR 
			stDeviceOpe.xPull_Hmi[5] OR 			
			stDeviceOpe.xPumpCal_Hmi OR 
			stDeviceOpe.xPush_Hmi[1] OR 
			stDeviceOpe.xPush_Hmi[2] OR 
			stDeviceOpe.xPush_Hmi[3] OR 			
			stDeviceOpe.xPush_Hmi[4] OR 			
			stDeviceOpe.xPush_Hmi[5] OR 						
			stDeviceOpe.xResetCalcoeffCal_Hmi OR 
			stDeviceOpe.xStop_Hmi;
_xAutoOpe:=	
						stDeviceOpe.xConfigure_Auto OR 
            stDeviceOpe.xFullSpeedPull_Auto OR 
            stDeviceOpe.xFullSpeedPush_Auto OR 
            stDeviceOpe.xPull_Auto[1] OR 
            stDeviceOpe.xPull_Auto[2] OR 			
            stDeviceOpe.xPull_Auto[3] OR 			
            stDeviceOpe.xPull_Auto[4] OR 			
            stDeviceOpe.xPull_Auto[5] OR 			
            stDeviceOpe.xPumpCal_Auto OR 
            stDeviceOpe.xPush_Auto[1] OR 
            stDeviceOpe.xPush_Auto[2] OR 			
            stDeviceOpe.xPush_Auto[3] OR 			
            stDeviceOpe.xPush_Auto[4] OR 			
            stDeviceOpe.xPush_Auto[5] OR 						
            stDeviceOpe.xStop_Auto;

METHOD PROTECTED AbortAction
VAR_INPUT
END_VAR
VAR_OUTPUT
	xComplete: BOOL;
  eERRORID: RudongPump_ERROR;
END_VAR
(*
* Cleaning
* => abort all running operation
* => if an NBS.RudongPump_ERROR codition is reached, set eERRORID to a Value rather then NBS.RudongPump_ERROR.No_ERROR 
*)
xComplete:=1;
eERRORID:=RudongPump_ERROR.No_ERROR;
END_METHOD

ACTION ACT_GetModbusAdr:
//
(*************************检测配置参数是否匹配成功*********************************)
IF stRunPara.iPumpType=RudongPump_PumpType.DFPluse THEN//DF600Plus/KF300系列
	_aMBAddr[1]:= 	stModbusAddress.iPumpType_Address									:=1000;
	_aMBAddr[2]:= 	stModbusAddress.iHosePipeType_Address							:=1001;	
	_aMBAddr[6]:=		stModbusAddress.iFluVolumeSet_Address							:=1002;
	_aMBAddr[7]:=		stModbusAddress.iRuntimeSet_Address								:=1004;
	//_aMBAddr[5]:=		stModbusAddress.iIntervalTime_Address							:=1006;
	_aMBAddr[9]:=		stModbusAddress.iCycleNumber_Address							:=1008;
	_aMBAddr[8]:=		stModbusAddress.iBackAngle_Address								:=1009;
	_aMBAddr[4]:=		stModbusAddress.iMoveDirection_Address						:=1010;
	_aMBAddr[3]:=		stModbusAddress.iStartStop_Address								:=1011;
	_aMBAddr[5]:=		stModbusAddress.iFullSpeedStartStop_Address				:=1012;
	_aMBAddr[10]:=	stModbusAddress.iModuleAddress_Address						:=2000;
	_aMBAddr[12]:=	stModbusAddress.iModuleStartStop_Address					:=2003;
	_aMBAddr[13]:=	stModbusAddress.iModuleRealFluVolumeSet_Address		:=2004;
	_aMBAddr[15]:=	stModbusAddress.iRecoveryCalCoefficient_Address		:=2007;	

ELSIF stRunPara.iPumpType=RudongPump_PumpType.F OR 
			stRunPara.iPumpType=RudongPump_PumpType.LabF1 OR
			stRunPara.iPumpType=RudongPump_PumpType.LabF3 OR
			stRunPara.iPumpType=RudongPump_PumpType.LabF4
THEN
	_aMBAddr[1]:= stModbusAddress.iPumpType_Address:=1000;
	_aMBAddr[2]:= stModbusAddress.iHosePipeType_Address:=1001;	
	_aMBAddr[6]:=	stModbusAddress.iFluVolumeSet_Address:=1015;
	_aMBAddr[7]:=	stModbusAddress.iRuntimeSet_Address:=1018;
	//_aMBAddr[5]:=	stModbusAddress.iIntervalTime_Address:=1021;
	_aMBAddr[9]:=	stModbusAddress.iCycleNumber_Address:=1023;
	_aMBAddr[8]:=	stModbusAddress.iBackAngle_Address:=1007;
	_aMBAddr[4]:=	stModbusAddress.iMoveDirection_Address:=1009;
	_aMBAddr[3]:=	stModbusAddress.iStartStop_Address:=1008;
	_aMBAddr[5]:=	stModbusAddress.iFullSpeedStartStop_Address:=1010;
	_aMBAddr[10]:=stModbusAddress.iModuleAddress_Address:=0;//等于0表示不写入
	_aMBAddr[12]:=stModbusAddress.iModuleStartStop_Address:=2003;
	_aMBAddr[13]:=stModbusAddress.iModuleRealFluVolumeSet_Address:=2004;
	_aMBAddr[15]:=stModbusAddress.iRecoveryCalCoefficient_Address:=2006;	

ELSIF stRunPara.iPumpType=RudongPump_PumpType.V THEN
	_aMBAddr[1]:= stModbusAddress.iPumpType_Address:=1000;
	_aMBAddr[2]:= stModbusAddress.iHosePipeType_Address:=1001;	
	_aMBAddr[6]:=	stModbusAddress.iFluVolumeSet_Address:=1015;
	_aMBAddr[7]:=	stModbusAddress.iRuntimeSet_Address:=1018;
	//_aMBAddr[5]:=	stModbusAddress.iIntervalTime_Address:=1021;
	_aMBAddr[9]:=	stModbusAddress.iCycleNumber_Address:=1023;
	_aMBAddr[8]:=	stModbusAddress.iBackAngle_Address:=1007;
	_aMBAddr[4]:=	stModbusAddress.iMoveDirection_Address:=1009;
	_aMBAddr[3]:=	stModbusAddress.iStartStop_Address:=1008;
	_aMBAddr[5]:=	stModbusAddress.iFullSpeedStartStop_Address:=1010;
	_aMBAddr[10]:=stModbusAddress.iModuleAddress_Address:=0;//等于0表示不写入
	_aMBAddr[12]:=stModbusAddress.iModuleStartStop_Address:=2003;
	_aMBAddr[13]:=stModbusAddress.iModuleRealFluVolumeSet_Address:=2004;
	_aMBAddr[15]:=stModbusAddress.iRecoveryCalCoefficient_Address:=2006;


END_IF

_aMBAddr[16]:=stModbusAddress.iStartStop_Address;
_aMBAddr[17]:=stModbusAddress.iModuleStartStop_Address;
END_ACTION

ACTION ACT_PumpPar:
//
(*************************检测配置参数是否匹配成功*********************************)
IF stRunPara.iPumpType=RudongPump_PumpType.DFPluse THEN
	//MiniPump泵头
	IF  stRunPara.iPumpTypeSet=RudongPump_PumpHeadType.MiniPump01 THEN
		st_IOData.O_PumpType:=0;//泵头值为0
			IF stRunPara.iHosePipeTypeSet=RudongPump_SoftPipeType.P13 THEN//13#软管
				st_IOData.O_HosePipeType:=13;//软管类型值13
				IF rFluVolumeSet*1000/135<0.1 THEN
					iMinRunTime:=	0.1;
				ELSE
					iMinRunTime:=	rFluVolumeSet*1000/135;
				END_IF
				iMaxRunTime:=	(rFluVolumeSet/0.45)*0.2;//最大流量(0.45微升/秒,0.0024ml/min)	
			ELSIF stRunPara.iHosePipeTypeSet=RudongPump_SoftPipeType.P14 THEN//14#软管
				st_IOData.O_HosePipeType:=14;
				IF rFluVolumeSet*1000/570<0.1 THEN
					iMinRunTime:=	0.1;
				ELSE
					iMinRunTime:=	rFluVolumeSet*1000/135;
				END_IF
				iMaxRunTime:=	(rFluVolumeSet/1.9)*0.2;	
			ELSIF stRunPara.iHosePipeTypeSet=RudongPump_SoftPipeType.P19 THEN//19#软管
				st_IOData.O_HosePipeType:=19;
				IF rFluVolumeSet*1000/1240<0.1 THEN
					iMinRunTime:=	0.1;
				ELSE
					iMinRunTime:=	rFluVolumeSet*1000/1240;
				END_IF
				iMaxRunTime:=	(rFluVolumeSet*1000/4.13)*0.2;		
			ELSIF stRunPara.iHosePipeTypeSet=RudongPump_SoftPipeType.P16 THEN//16#软管
				st_IOData.O_HosePipeType:=16;
				IF rFluVolumeSet*1000/1880<0.1 THEN
					iMinRunTime:=	0.1;
				ELSE
					iMinRunTime:=	rFluVolumeSet*1000/1880;
				END_IF
				iMaxRunTime:=	(rFluVolumeSet*1000/6.28)*0.2;	
			ELSIF stRunPara.iHosePipeTypeSet=RudongPump_SoftPipeType.P25 THEN//25#软管
				st_IOData.O_HosePipeType:=25;
				IF rFluVolumeSet*1000/3100<0.1 THEN
					iMinRunTime:=	0.1;
				ELSE
					iMinRunTime:=	rFluVolumeSet*1000/3100;
				END_IF
				iMaxRunTime:=	(rFluVolumeSet*1000/10.33)*0.2;			
		ELSE
				eERRORID:=RudongPump_ERROR.FLT_CONFIGURE_PARA;		
		END_IF
	//UD15
	ELSIF  stRunPara.iPumpTypeSet=RudongPump_PumpHeadType.UD15 THEN
		st_IOData.O_PumpType:=1;//泵头值为0
			IF stRunPara.iHosePipeTypeSet=RudongPump_SoftPipeType.P16 THEN//16#软管
				st_IOData.O_HosePipeType:=16;
				IF rFluVolumeSet*1000/4000<0.1 THEN
					iMinRunTime:=	0.1;
				ELSE
					iMinRunTime:=	rFluVolumeSet*1000/4000;
				END_IF
				iMaxRunTime:=	(rFluVolumeSet*1000/13.33)*0.2;		
			ELSIF stRunPara.iHosePipeTypeSet=RudongPump_SoftPipeType.P17 THEN//17#软管
				st_IOData.O_HosePipeType:=17;
				IF rFluVolumeSet*1000/15000<0.1 THEN
					iMinRunTime:=	0.1;
				ELSE
					iMinRunTime:=	rFluVolumeSet*1000/15000;
				END_IF
				iMaxRunTime:=	(rFluVolumeSet*1000/50)*0.2;	
			ELSIF stRunPara.iHosePipeTypeSet=RudongPump_SoftPipeType.P25 THEN//25#软管
				st_IOData.O_HosePipeType:=25;
				IF rFluVolumeSet*1000/8000<0.1 THEN
					iMinRunTime:=	0.1;
				ELSE
					iMinRunTime:=	rFluVolumeSet*1000/8000;
				END_IF
				iMaxRunTime:=	(rFluVolumeSet*1000/26.66)*0.2;			
		ELSE
				eERRORID:=RudongPump_ERROR.FLT_CONFIGURE_PARA;		
		END_IF
	//HandyPump01泵头
ELSIF  stRunPara.iPumpTypeSet=RudongPump_PumpHeadType.HandyPump01 THEN
 			IF stRunPara.iHosePipeTypeSet=RudongPump_SoftPipeType.P13 THEN//13#软管,三滚轮
				IF rFluVolumeSet*1000/155<0.1 THEN
					iMinRunTime:=	0.1;
				ELSE
					iMinRunTime:=	rFluVolumeSet*1000/155;
				END_IF
				iMaxRunTime:=	(rFluVolumeSet*1000/0.51)*0.2;	
		
	(*	IF stRunPara.iHosePipeTypeSet=RudongPump_SoftPipeType.P13 THEN//13#软管,三滚轮
			iMinRunTime:=	(rFluVolumeSet/10)*60;
			iMaxRunTime:=	(rFluVolumeSet/0.0033)*60;	
		ELSIF stRunPara.iHosePipeTypeSet=RudongPump_SoftPipeType.P14 THEN//14#软管,三滚轮
			iMinRunTime:=	(rFluVolumeSet/56)*60;
			iMaxRunTime:=	(rFluVolumeSet/0.0187)*60;		
		ELSIF stRunPara.iHosePipeTypeSet=RudongPump_SoftPipeType.P19 THEN//19#软管,三滚轮
			iMinRunTime:=	(rFluVolumeSet/111)*60;
			iMaxRunTime:=	(rFluVolumeSet/0.0371)*60;
		ELSIF stRunPara.iHosePipeTypeSet=RudongPump_SoftPipeType.P16 THEN//16#软管,三滚轮
			iMinRunTime:=	(rFluVolumeSet/190)*60;
			iMaxRunTime:=	(rFluVolumeSet/0.0636)*60;		
		ELSIF stRunPara.iHosePipeTypeSet=RudongPump_SoftPipeType.P25 THEN//25#软管,三滚轮
			iMinRunTime:=	(rFluVolumeSet/365)*60;
			iMaxRunTime:=	(rFluVolumeSet/0.1219)*60;
	*)
		ELSE
				eERRORID:=RudongPump_ERROR.FLT_CONFIGURE_PARA;						
		END_IF
	END_IF
ELSE
		eERRORID:=RudongPump_ERROR.FLT_CONFIGURE_PARA;
END_IF


(*
//MiniPump01泵头
IF  stRunPara.iPumpTypeSet=RudongPump_PumpHeadType.MiniPump01 THEN
		IF stRunPara.iHosePipeTypeSet=RudongPump_SoftPipeType.P13 THEN//13#软管
			iMinRunTime:=	(rFluVolumeSet/8)*60;//最大流量(135微升/秒,8.28ml/min)
			iMaxRunTime:=	(rFluVolumeSet/0.45)*60;//最大流量(0.45微升/秒,0.0024ml/min)	
		ELSIF stRunPara.iHosePipeTypeSet=RudongPump_SoftPipeType.P14 THEN//14#软管
			iMinRunTime:=	(rFluVolumeSet/33)*60;
			iMaxRunTime:=	(rFluVolumeSet/1.9)*60;
		ELSIF stRunPara.iHosePipeTypeSet=RudongPump_SoftPipeType.P19 THEN//19#软管
			iMinRunTime:=	(rFluVolumeSet/77)*60;
			iMaxRunTime:=	(rFluVolumeSet/4.13)*60;	
		ELSIF stRunPara.iHosePipeTypeSet=RudongPump_SoftPipeType.P16 THEN//16#软管
			iMinRunTime:=	(rFluVolumeSet/114)*60;
			iMaxRunTime:=	(rFluVolumeSet/6.28)*60;	
		ELSIF stRunPara.iHosePipeTypeSet=RudongPump_SoftPipeType.P25 THEN//25#软管
			iMinRunTime:=	(rFluVolumeSet/190)*60;
			iMaxRunTime:=	(rFluVolumeSet/10.33)*60;		
		ELSIF stRunPara.iHosePipeTypeSet=RudongPump_SoftPipeType.P1_1 THEN//1x1#软管
			iMinRunTime:=	(rFluVolumeSet/15)*60;
			iMaxRunTime:=	(rFluVolumeSet/4.5)*60;	
		ELSIF stRunPara.iHosePipeTypeSet=RudongPump_SoftPipeType.P2_1 THEN//2x1#软管
			iMinRunTime:=	(rFluVolumeSet/54)*60;
			iMaxRunTime:=	(rFluVolumeSet/4.5)*60;		
		ELSIF stRunPara.iHosePipeTypeSet=RudongPump_SoftPipeType.P2_5_1 THEN//2.5x1#软管
			iMinRunTime:=	(rFluVolumeSet/76)*60;
			iMaxRunTime:=	(rFluVolumeSet/5)*60;		
		ELSIF stRunPara.iHosePipeTypeSet=RudongPump_SoftPipeType.P3_1 THEN//3x1#软管
			iMinRunTime:=	(rFluVolumeSet/108)*60;
			iMaxRunTime:=	(rFluVolumeSet/5)*60;
	ELSE
			eERRORID:=RudongPump_ERROR.FLT_CONFIGURE_PARA;		
	END_IF		
	
//MiniPump02泵头
ELSIF  stRunPara.iPumpTypeSet=RudongPump_PumpHeadType.MiniPump02 THEN
	IF stRunPara.iHosePipeTypeSet=RudongPump_SoftPipeType.P1_1 THEN//1x1#软管
		iMinRunTime:=	(rFluVolumeSet/15.01)*60;
		iMaxRunTime:=	(rFluVolumeSet/0.005)*60;	
	ELSIF stRunPara.iHosePipeTypeSet=RudongPump_SoftPipeType.P2_1 THEN//2x1#软管
		iMinRunTime:=	(rFluVolumeSet/54.63)*60;
		iMaxRunTime:=	(rFluVolumeSet/0.018)*60;		
	ELSIF stRunPara.iHosePipeTypeSet=RudongPump_SoftPipeType.P2_5_1 THEN//2.5x1#软管
		iMinRunTime:=	(rFluVolumeSet/76.84)*60;
		iMaxRunTime:=	(rFluVolumeSet/0.0256)*60;
	ELSE
			eERRORID:=RudongPump_ERROR.FLT_CONFIGURE_PARA;						
	END_IF	

//HandyPump01泵头
ELSIF  stRunPara.iPumpTypeSet=RudongPump_PumpHeadType.HandyPump01 THEN
	IF stRunPara.iHosePipeTypeSet=RudongPump_SoftPipeType.P13 THEN//13#软管,三滚轮
		iMinRunTime:=	(rFluVolumeSet/10)*60;
		iMaxRunTime:=	(rFluVolumeSet/0.0033)*60;	
	ELSIF stRunPara.iHosePipeTypeSet=RudongPump_SoftPipeType.P14 THEN//14#软管,三滚轮
		iMinRunTime:=	(rFluVolumeSet/56)*60;
		iMaxRunTime:=	(rFluVolumeSet/0.0187)*60;		
	ELSIF stRunPara.iHosePipeTypeSet=RudongPump_SoftPipeType.P19 THEN//19#软管,三滚轮
		iMinRunTime:=	(rFluVolumeSet/111)*60;
		iMaxRunTime:=	(rFluVolumeSet/0.0371)*60;
	ELSIF stRunPara.iHosePipeTypeSet=RudongPump_SoftPipeType.P16 THEN//16#软管,三滚轮
		iMinRunTime:=	(rFluVolumeSet/190)*60;
		iMaxRunTime:=	(rFluVolumeSet/0.0636)*60;		
	ELSIF stRunPara.iHosePipeTypeSet=RudongPump_SoftPipeType.P25 THEN//25#软管,三滚轮
		iMinRunTime:=	(rFluVolumeSet/365)*60;
		iMaxRunTime:=	(rFluVolumeSet/0.1219)*60;
	ELSE
			eERRORID:=RudongPump_ERROR.FLT_CONFIGURE_PARA;						
	END_IF

//HandyPump02泵头
ELSIF  stRunPara.iPumpTypeSet=RudongPump_PumpHeadType.HandyPump02 THEN
	IF stRunPara.iHosePipeTypeSet=RudongPump_SoftPipeType.P13 THEN//13#软管,三滚轮
		iMinRunTime:=	(rFluVolumeSet/10)*60;
		iMaxRunTime:=	(rFluVolumeSet/0.0033)*60;	
	ELSIF stRunPara.iHosePipeTypeSet=RudongPump_SoftPipeType.P14 THEN//14#软管,三滚轮
		iMinRunTime:=	(rFluVolumeSet/56)*60;
		iMaxRunTime:=	(rFluVolumeSet/0.0187)*60;		
	ELSIF stRunPara.iHosePipeTypeSet=RudongPump_SoftPipeType.P19 THEN//19#软管,三滚轮
		iMinRunTime:=	(rFluVolumeSet/111)*60;
		iMaxRunTime:=	(rFluVolumeSet/0.0371)*60;
	ELSIF stRunPara.iHosePipeTypeSet=RudongPump_SoftPipeType.P16 THEN//16#软管,三滚轮
		iMinRunTime:=	(rFluVolumeSet/190)*60;
		iMaxRunTime:=	(rFluVolumeSet/0.0636)*60;	
	ELSE
			eERRORID:=RudongPump_ERROR.FLT_CONFIGURE_PARA;							
	END_IF

//EasyPumpI_III泵头,单通道
ELSIF  stRunPara.iPumpTypeSet=RudongPump_PumpHeadType.EasyPumpI_III THEN
	IF stRunPara.iHosePipeTypeSet=RudongPump_SoftPipeType.P13 THEN//13#软管
		iMinRunTime:=	(rFluVolumeSet/32)*60;
		iMaxRunTime:=	(rFluVolumeSet/0.0053)*60;	
	ELSIF stRunPara.iHosePipeTypeSet=RudongPump_SoftPipeType.P14 THEN//14#软管
		iMinRunTime:=	(rFluVolumeSet/162)*60;
		iMaxRunTime:=	(rFluVolumeSet/0.027)*60;		
	ELSIF stRunPara.iHosePipeTypeSet=RudongPump_SoftPipeType.P19 THEN//19#软管
		iMinRunTime:=	(rFluVolumeSet/330)*60;
		iMaxRunTime:=	(rFluVolumeSet/0.055)*60;
	ELSIF stRunPara.iHosePipeTypeSet=RudongPump_SoftPipeType.P16 THEN//16#软管
		iMinRunTime:=	(rFluVolumeSet/560)*60;
		iMaxRunTime:=	(rFluVolumeSet/0.093)*60;	
	ELSIF stRunPara.iHosePipeTypeSet=RudongPump_SoftPipeType.P25 THEN//25#软管
		iMinRunTime:=	(rFluVolumeSet/1180)*60;
		iMaxRunTime:=	(rFluVolumeSet/0.197)*60;	
	ELSIF stRunPara.iHosePipeTypeSet=RudongPump_SoftPipeType.P17 THEN//17#软管
		iMinRunTime:=	(rFluVolumeSet/2000)*60;
		iMaxRunTime:=	(rFluVolumeSet/0.333)*60;	
	ELSIF stRunPara.iHosePipeTypeSet=RudongPump_SoftPipeType.P18 THEN//18#软管
		iMinRunTime:=	(rFluVolumeSet/2580)*60;
		iMaxRunTime:=	(rFluVolumeSet/0.430)*60;	
	ELSE
			eERRORID:=RudongPump_ERROR.FLT_CONFIGURE_PARA;							
	END_IF

//EasyPumpII_IV泵头,单通道
ELSIF  stRunPara.iPumpTypeSet=RudongPump_PumpHeadType.EasyPumpII_IV THEN
	IF stRunPara.iHosePipeTypeSet=RudongPump_SoftPipeType.P15 THEN//15#软管
		iMinRunTime:=	(rFluVolumeSet/1080)*60;
		iMaxRunTime:=	(rFluVolumeSet/0.0180)*60;	
	ELSIF stRunPara.iHosePipeTypeSet=RudongPump_SoftPipeType.P24 THEN//24#软管
		iMinRunTime:=	(rFluVolumeSet/1640)*60;
		iMaxRunTime:=	(rFluVolumeSet/0.273)*60;		
	ELSIF stRunPara.iHosePipeTypeSet=RudongPump_SoftPipeType.P35 THEN//35#软管
		iMinRunTime:=	(rFluVolumeSet/2300)*60;
		iMaxRunTime:=	(rFluVolumeSet/0.383)*60;
	ELSIF stRunPara.iHosePipeTypeSet=RudongPump_SoftPipeType.P36 THEN//36#软管
		iMinRunTime:=	(rFluVolumeSet/3100)*60;
		iMaxRunTime:=	(rFluVolumeSet/0.517)*60;	
	ELSE
			eERRORID:=RudongPump_ERROR.FLT_CONFIGURE_PARA;							
	END_IF

//EasyPumpV_VI泵头,双通道
ELSIF  stRunPara.iPumpTypeSet=RudongPump_PumpHeadType.EasyPumpV_VI THEN
		IF stRunPara.iHosePipeTypeSet=RudongPump_SoftPipeType.P13 THEN//13#软管
		iMinRunTime:=	(rFluVolumeSet/32)*60;
		iMaxRunTime:=	(rFluVolumeSet/0.0053)*60;	
	ELSIF stRunPara.iHosePipeTypeSet=RudongPump_SoftPipeType.P14 THEN//14#软管
		iMinRunTime:=	(rFluVolumeSet/162)*60;
		iMaxRunTime:=	(rFluVolumeSet/0.0027)*60;		
	ELSIF stRunPara.iHosePipeTypeSet=RudongPump_SoftPipeType.P19 THEN//19#软管
		iMinRunTime:=	(rFluVolumeSet/330)*60;
		iMaxRunTime:=	(rFluVolumeSet/0.0055)*60;
	ELSIF stRunPara.iHosePipeTypeSet=RudongPump_SoftPipeType.P16 THEN//16#软管
		iMinRunTime:=	(rFluVolumeSet/560)*60;
		iMaxRunTime:=	(rFluVolumeSet/0.093)*60;		
	ELSIF stRunPara.iHosePipeTypeSet=RudongPump_SoftPipeType.P25 THEN//25#软管
		iMinRunTime:=	(rFluVolumeSet/1180)*60;
		iMaxRunTime:=	(rFluVolumeSet/0.197)*60;
	ELSE
			eERRORID:=RudongPump_ERROR.FLT_CONFIGURE_PARA;							
	END_IF
	
END_IF


END_IF

*)
		


//参数超出范围报错	
IF rFluVolumeSet<>0 THEN
	IF rRuntimeSet<iMinRunTime OR rRuntimeSet>iMaxRunTime OR  iMaxRunTime<iMinRunTime THEN
		eERRORID:=RudongPump_ERROR.FLT_CONFIGURE_PARA;
	END_IF
END_IF
END_ACTION

ACTION ACTMap:
//进行数据刷新(判断疏浚地址是否有效)

//1,泵头类型
	_aAddr[1,1]:=st_IOData.O_PumpType;
//2,软管类型	
	_aAddr[2,1]:=st_IOData.O_HosePipeType;
//3,启停控制	
	_aAddr[3,1]:=st_IOData.O_ControlSet;
//4,方向控制	
	_aAddr[4,1]:=st_IOData.O_DirectionSet;
//5,全速控制	
	_aAddr[5,1]:=st_IOData.O_FullSpeedControl;	
//6,液量设定	


//8,回吸角度	
	_aAddr[8,1]:=st_IOData.O_BackAngle;    /////////
//9,重复次数	
	_aAddr[9,1]:=st_IOData.O_CycleNumber;
//10,灌装单元地址
	_aAddr[10,1]:=st_IOData.O_ModuleAddress;	
//11,灌装单元速度____________________
	SysMemCpy(ADR(_aAddr[11,1]),ADR(st_IOData.O_ModuleSpeed),4);
	_wModuleSpeedSetTemp := TO_WORD(_aAddr[11,1]);
	_aAddr[11,1] := _aAddr[11,2];
	_aAddr[11,2] := TO_INT(_wModuleSpeedSetTemp);			
//12,灌装单元启停
	_aAddr[12,1]:=st_IOData.O_ModuleStart;	
//13,实际灌装液量
	SysMemCpy(ADR(_aAddr[13,1]),ADR(st_IOData.O_ModuleRealVolume),4);
	_wModuleRealVolumeTemp := TO_WORD(_aAddr[13,1]);
	_aAddr[13,1] := _aAddr[13,2];
	_aAddr[13,2] := TO_INT(_wModuleRealVolumeTemp);		
//14,灌装液量微调__________________
	_aAddr[14,1]:=st_IOData.O_ModuleMicroReg;	
//15,恢复校准系数
	_aAddr[15,1]:=st_IOData.O_ResetCalcoeff;
//16,Run信号______________
	SysMemCpy(ADR(st_IOData.I_RunSignal),ADR(_aAddr[16,1]),2);	
//17,校准信号
	SysMemCpy(ADR(st_IOData.I_CalSignal),ADR(_aAddr[17,1]),2);

	

xRunning:=(st_IOData.I_RunSignal=1) OR (st_IOData.I_CalSignal=1);//运行信号
iPumpType:=RudongPump_PumpType.DFPluse;//蠕动泵类型
_fResetCheck(CLK:=xResetRequest);
xRdyCmd := eState = STATE.DORMANT AND eERRORID = RudongPump_ERROR.No_ERROR;//检测是否允许指令控制(初始状态，没有报警发生)
_rInit(CLK:= xIniting);//检测是否是初始化中，如果是的去切换模式
IF _rInit.Q
THEN
 eState := STATE.RESETING;
END_IF 
xDone:=_xDone AND xExecute;
xError:=eState=STATE.INERROR;//报错发生
(**********************************检测是否有模式切换********************************)
_rManual(CLK:=xAutoMode);
_fManual(CLK:=xAutoMode);
IF eState <> STATE.DORMANT//只有在运行的时候，才会检测是否有模式切换发生
THEN
	IF _rManual.Q OR _fManual.Q
	THEN
		_xModeChange := TRUE;//通知系统有模式切换发生
	END_IF	
END_IF
IF eState = STATE.DORMANT//要是待机模式下，切换模式，是不会起作用的
THEN
	_xModeChange := FALSE;
END_IF
END_ACTION

METHOD PROTECTED CmdCalParWrite
VAR_OUTPUT
	xComplete: BOOL;
END_VAR
// return the real actual fault number
IF eERRORID <> RudongPump_ERROR.No_ERROR
THEN
  RETURN;  
END_IF

CASE _diCmdState OF	
		
	0://单元实际液量设定
		_tonDelay(IN:= TRUE,pt:=T#20MS);//保证执行的是最新的一次
		st_IOData.O_ModuleRealVolume := iModuleRealVolume	;	
			st_IOData.O_FluVolumeSet := rFluVolumeSet	;	
		IF _tonDelay.Q
		THEN	
			IF ABS(st_IOData.O_ModuleRealVolume-st_IOData.O_FluVolumeSet)<(st_IOData.O_FluVolumeSet*0.5) THEN//误差不能超过0.3ml
				_aExecute[13] := TRUE;//
				//复位定时器
				_tonDelay(IN:=FALSE);
				_tonCmdTimeout(in:=FALSE);
				_tonTimeout(in:=FALSE);
				_diCmdState := _diCmdState+1;//切换状态										
			ELSE
				eERRORID := RudongPump_ERROR.FLT_PumpCal_OverFlow;//误差过大
				_diCmdState := 999;
			END_IF	
		END_IF
		
	1://等待单元实际液量设定被响应
		IF NOT _aExecute[13]//
		THEN		
				_tonTimeout(in:=FALSE);
				_tonDelay(IN:=FALSE);
				_tonCmdTimeout(IN:= FALSE); 
				_diCmdState := _diCmdState+1;//切换状态	
		END_IF	
		IF _rxstate=999
		THEN
			eERRORID := RudongPump_ERROR.FLT_CMD_TIMEOUT;		
			_diCmdState := 999;
		END_IF		

	2://
		xComplete := TRUE; 
		
	ELSE
		;	
END_CASE
END_METHOD

METHOD PROTECTED CmdCalReset
VAR_OUTPUT
	xComplete: BOOL;
END_VAR
// return the real actual fault number
IF eERRORID <> RudongPump_ERROR.No_ERROR
THEN
  RETURN;  
END_IF

CASE _diCmdState OF					
	0://发送灌装系数复位指令
		_tonDelay(IN:= TRUE,pt:=T#20MS);//保证执行的是最新的一次
		st_IOData.O_ResetCalcoeff := 1	;	
		IF _tonDelay.Q
		THEN	
			_aExecute[15] := TRUE;//	
			//复位定时器
			_tonDelay(IN:=FALSE);
			_tonCmdTimeout(in:=FALSE);
			_tonTimeout(in:=FALSE);
			_diCmdState := _diCmdState+1;//切换状态
		END_IF
		
	1://等待灌装启动被响应
		IF NOT _aExecute[15]//
		THEN		
				_tonTimeout(in:=FALSE);
				_tonDelay(IN:=FALSE);
				_tonCmdTimeout(IN:= FALSE); 
				_diCmdState := _diCmdState+1;//切换状态	
		END_IF	
		IF _rxState=999
		THEN
			eERRORID := RudongPump_ERROR.FLT_CMD_TIMEOUT;		
			_diCmdState := 999;
		END_IF	

	2://
		xComplete := TRUE; 
		
	ELSE
		;	
END_CASE
END_METHOD

METHOD PROTECTED CmdPumpCal
VAR_OUTPUT
	xComplete: BOOL;
END_VAR
// return the real actual fault number
IF eERRORID <> RudongPump_ERROR.No_ERROR
THEN
  RETURN;  
END_IF

CASE _diCmdState OF	
	0://检查参数	  	
		IF xNeedConfigurePara
		THEN
			_tonDelay(IN:= TRUE,pt:=T#25MS);//保证执行的是最新的一次
			IF _tonDelay.Q
			THEN	
				//复位定时器
				_tonDelay(IN:=FALSE);
				_tonCmdTimeout(in:=FALSE);
				_tonTimeout(in:=FALSE);
				_diCmdState := _diCmdState+1;//切换状态
			END_IF
		ELSE//直接启动就好
			//复位定时器
			_tonDelay(IN:=FALSE);
			_tonCmdTimeout(in:=FALSE);
			_tonTimeout(in:=FALSE);
			_diCmdState := 8;//切换状态
		END_IF	
		//检测流量转速是否在0.1rpm - 600rpm
		IF 	rRuntimeSet = 0 
		THEN 
			eERRORID := RudongPump_ERROR.FLT_FLUVOLUM_TIME_PARA;		
			_diCmdState := 999;
		ELSE
			_rSetSpeed := rFluVolumeSet * 60.0 / rSpeedRatio / rRuntimeSet;
			IF _rSetSpeed >= 0.001 AND _rSetSpeed <= 600
			THEN
				;
			ELSE
				eERRORID := RudongPump_ERROR.FLT_FLUVOLUM_TIME_PARA;		
				_diCmdState := 999;
			END_IF
		END_IF						
	1://等待定时定量模式被响应			
		_tonTimeout(in:=FALSE);
		_tonDelay(IN:=FALSE);
		_tonCmdTimeout(IN:= FALSE);    
		_diCmdState := _diCmdState+1;//切换状态	
		IF _rxstate=999
		THEN
			eERRORID := RudongPump_ERROR.FLT_CMD_TIMEOUT;		
			_diCmdState := 999;
		END_IF
//发送虚假定量时间		
	2://定量时间设定		
		_tonDelay(IN:= TRUE,pt:=T#25MS);//保证执行的是最新的一次
		st_IOData.O_RuntimeSet := 5.0	;	//保证电机转速不会超
		IF _tonDelay.Q
		THEN	
			_aExecute[7] := TRUE;//启动夹紧控制数据发送	
			//复位定时器
			_tonDelay(IN:=FALSE);
			_tonCmdTimeout(in:=FALSE);
			_tonTimeout(in:=FALSE);
			_diCmdState := _diCmdState+1;//切换状态
		END_IF
	3://等待定量时间设定被响应
		IF NOT _aExecute[7]//
		THEN	
			_tonDelay(IN:=TRUE,PT:= T#50MS);
			IF _tonDelay.Q
			THEN							
				_tonTimeout(in:=FALSE);
				_tonDelay(IN:=FALSE);
				_tonCmdTimeout(IN:= FALSE);    
				_diCmdState := _diCmdState+1;//切换状态
			END_IF					
		END_IF	
		IF _rxstate=999
		THEN
			eERRORID := RudongPump_ERROR.FLT_CMD_TIMEOUT;		
			_diCmdState := 999;
		END_IF		
		
		
//传递液量参数		
	4://		
		_tonDelay(IN:= TRUE,pt:=T#25MS);//保证执行的是最新的一次
		st_IOData.O_FluVolumeSet := rFluVolumeSet	;	
		IF _tonDelay.Q
		THEN	
			_aExecute[6] := TRUE;//启动夹紧控制数据发送	
			//复位定时器
			_tonDelay(IN:=FALSE);
			_tonCmdTimeout(in:=FALSE);
			_tonTimeout(in:=FALSE);
			_diCmdState := _diCmdState+1;//切换状态
		END_IF	  
	5://等待流量设定结束
		IF NOT _aExecute[6]//
		THEN	
			_tonDelay(IN:=TRUE,PT:= T#50MS);
			IF _tonDelay.Q
			THEN			
				_tonTimeout(in:=FALSE);
				_tonDelay(IN:=FALSE);
				_tonCmdTimeout(IN:= FALSE);    
				_diCmdState := _diCmdState+1;//切换状态
			END_IF				
		END_IF	
		IF _rxstate=999
		THEN
			eERRORID := RudongPump_ERROR.FLT_CMD_TIMEOUT;		
			_diCmdState := 999;
		END_IF

//传递实际定量时间		
	6://定量时间设定		
		_tonDelay(IN:= TRUE,pt:=T#25MS);//保证执行的是最新的一次
		st_IOData.O_RuntimeSet := rRuntimeSet	;	
		IF _tonDelay.Q
		THEN	
			_aExecute[7] := TRUE;//启动夹紧控制数据发送	
			//复位定时器
			_tonDelay(IN:=FALSE);
			_tonCmdTimeout(in:=FALSE);
			_tonTimeout(in:=FALSE);
			_diCmdState := _diCmdState+1;//切换状态
		END_IF
		
	7://等待定量时间设定被响应
		IF NOT _aExecute[7]//
		THEN			
			_tonDelay(IN:=TRUE,PT:= T#50MS);
			IF _tonDelay.Q
			THEN			
				_tonTimeout(in:=FALSE);
				_tonDelay(IN:=FALSE);
				_tonCmdTimeout(IN:= FALSE);    
				_diCmdState := _diCmdState+1;//切换状态	
			END_IF				
		END_IF	
		IF _rxstate=999
		THEN
			eERRORID := RudongPump_ERROR.FLT_CMD_TIMEOUT;		
			_diCmdState := 999;
		END_IF	
		
	8://方向设定		
		_tonDelay(IN:= ( eCmd = RudongPump_CMD.Cmd_CalPump ) ,pt:=T#20MS);//保证执行的是最新的一次
		st_IOData.O_DirectionSet := iDirectionSet	;			
		IF _tonDelay.Q
		THEN	
			_aExecute[4] := TRUE;//启动夹紧控制数据发送	
			//复位定时器
			_tonDelay(IN:=FALSE);
			_tonCmdTimeout(in:=FALSE);
			_tonTimeout(in:=FALSE);
			_diCmdState := _diCmdState+1;//切换状态
		END_IF
		
	9://等待方向设定被响应
		IF NOT _aExecute[4]//
		THEN		
			_diCmdState := _diCmdState +1; 
			_tonDelay(IN:=FALSE);
			_tonCmdTimeout(in:=FALSE);
			_tonTimeout(in:=FALSE);
		END_IF	
		IF _rxstate=999
		THEN
			eERRORID := RudongPump_ERROR.FLT_CMD_TIMEOUT;		
			_diCmdState := 999;
		END_IF	
		
	10://重复次数设定		
		_tonDelay(IN:= TRUE,pt:=T#25MS);//保证执行的是最新的一次
		st_IOData.O_CycleNumber := iCycleNumber	;	
		IF _tonDelay.Q
		THEN	
			_aExecute[9] := TRUE;//启动夹紧控制数据发送	
			//复位定时器
			_tonDelay(IN:=FALSE);
			_tonCmdTimeout(in:=FALSE);
			_tonTimeout(in:=FALSE);
			_diCmdState := _diCmdState+1;//切换状态
		END_IF
		
	11://等待重复次数设定被响应
		IF NOT _aExecute[9]//
		THEN
			_tonDelay(IN:=TRUE,PT:= T#50MS);
			IF _tonDelay.Q
			THEN		
				_tonTimeout(in:=FALSE);
				_tonDelay(IN:=FALSE);
				_tonCmdTimeout(IN:= FALSE); 
				_diCmdState := _diCmdState+1;//切换状态
			END_IF				
		END_IF	
		IF _rxState=999
		THEN
			eERRORID := RudongPump_ERROR.FLT_CMD_TIMEOUT;		
			_diCmdState := 999;
		END_IF		
		
	12://单元地址设定
		_tonDelay(IN:= TRUE,pt:=T#20MS);//保证执行的是最新的一次
		st_IOData.O_ModuleAddress := iModuleAdress	;
		//st_IOData.O_ModuleSpeed := iModuleSpeed	;	
		IF _tonDelay.Q
		THEN	
			_aExecute[10] := TRUE;//	
			//复位定时器
			_tonDelay(IN:=FALSE);
			_tonCmdTimeout(in:=FALSE);
			_tonTimeout(in:=FALSE);
			_diCmdState := _diCmdState+1;//切换状态
		END_IF
		
	13://等待单元地址设定被响应
	IF iPumpType=RudongPump_PumpType.DFPluse THEN	
		IF NOT _aExecute[10]//
		THEN		
			_tonDelay(IN:=TRUE,PT:= T#50MS);
			IF _tonDelay.Q
			THEN		
				_tonTimeout(in:=FALSE);
				_tonDelay(IN:=FALSE);
				_tonCmdTimeout(IN:= FALSE); 
				_diCmdState := _diCmdState+1;//切换状态
			END_IF				
		END_IF	
		IF _rxState=999
		THEN
			eERRORID := RudongPump_ERROR.FLT_CMD_TIMEOUT;		
			_diCmdState := 999;
		END_IF
	ELSE
		_diCmdState := 15;	
	END_IF	
		
	14://单元速度设定
	IF st_IOData.O_RunModeSet =1	THEN//如果是定量模式，需要设置速度
		_tonDelay(IN:= TRUE,pt:=T#20MS);//保证执行的是最新的一次
		st_IOData.O_ModuleSpeed := iModuleSpeed	;	
		IF _tonDelay.Q
		THEN	
			_aExecute[11] := TRUE;//	
			//复位定时器
			_tonDelay(IN:=FALSE);
			_tonCmdTimeout(in:=FALSE);
			_tonTimeout(in:=FALSE);
			_diCmdState := _diCmdState+1;//切换状态
		END_IF
	ELSE
		_diCmdState :=16;//如果是定时定量模式，则不需要设置速度
	END_IF	
	
	15://等待单元速度设定被响应
		_iNGCount :=0;
		IF NOT _aExecute[11]//
		THEN		
				_tonTimeout(in:=FALSE);
				_tonDelay(IN:=FALSE);
				_tonCmdTimeout(IN:= FALSE); 
				_diCmdState := _diCmdState+1;//切换状态
		END_IF	
		IF _rxState=999
		THEN
			eERRORID := RudongPump_ERROR.FLT_CMD_TIMEOUT;		
			_diCmdState := 999;
		END_IF		
		
	16://复位	
		st_IOData.O_ModuleStart := 0	;
		_aExecute[12] := FALSE;//		
		_diCmdState := _diCmdState+1;//切换状态
		
	17://灌装启动
		_tonDelay(IN:= TRUE,pt:=T#20MS);//保证执行的是最新的一次
		st_IOData.O_ModuleStart := 1	;	
		IF _tonDelay.Q
		THEN	
			_aExecute[12] := TRUE;//	
			//复位定时器
			_tonDelay(IN:=FALSE);
			_tonCmdTimeout(in:=FALSE);
			_tonTimeout(in:=FALSE);
			_diCmdState := _diCmdState+1;//切换状态
		END_IF
		
	18://等待启动被响应						
		IF  NOT _aExecute[12] THEN
			_tonDelay(IN:= TRUE ,pt:=T#100MS);//等待蠕动泵运行
			IF _tonDelay.Q
			THEN
				_tonDelay(IN:=FALSE);
				_tonCmdTimeout(in:=FALSE);
				_tonTimeout(in:=FALSE);
				_diCmdState := _diCmdState+1;
			END_IF			
		END_IF	
		IF _rxState=999
		THEN
			eERRORID := RudongPump_ERROR.FLT_CMD_TIMEOUT;		
			_diCmdState := 999;
		END_IF		
	19://读取运行状态
		_tonCmdTimeout(in:=FALSE);
		_tonDelay(IN:=FALSE); 
		_tonTimeout(in:=TRUE,pt:=T#10S);//设置超时时间 
		_aExecute[17] := TRUE;//触发读取反馈数据  
		_diCmdState := _diCmdState +1; 	
 
	20://等待状态响应
		_tonTimeout(in:=TRUE,pt:=T#10S); 
	  //进行数据刷新  
	  IF NOT _aExecute[17] //等待读取数据完成
	  THEN
	    _tonDelay(IN:= TRUE,pt:=T#40MS);//设置刷新周期	  
	    //松开成功判定
	    IF st_IOData.I_CalSignal = 0
	    THEN
				_tonCmdTimeout(in:=FALSE);
				_tonDelay(IN:= FALSE);
				_tonTimeout(in:=FALSE);  
				_diCmdState := _diCmdState+1;
	    END_IF 	  
			IF _tonDelay.Q
			THEN
				 _diCmdState := _diCmdState - 1;//回到上一步重新进行状态刷新
			END_IF
			IF _rxState=999//
			THEN
				eERRORID := eERRORID := RudongPump_ERROR.FLT_CMD_TIMEOUT;
				_diCmdState := 999;
			END_IF
			IF _tonTimeout.Q//
			THEN
				IF eCmd = RudongPump_CMD.Cmd_Push
				THEN
					eERRORID := RudongPump_ERROR.FLT_PUSH_TIMEOUT;		
				END_IF
				IF eCmd = RudongPump_CMD.Cmd_Pull 
				THEN
					eERRORID := RudongPump_ERROR.FLT_PULL_TIMEOUT;			
				END_IF	
			 _diCmdState := 999;
			END_IF
  	END_IF 		
(*
	21://等待接液完成
		IF (st_IOData.I_CalSignal=0) AND (stDeviceOpe.xPumpCal_Hmi OR stDeviceOpe.xPumpCal_Auto) AND NOT _xCheckModbusRun THEN
			_diCmdState := _diCmdState+1;//切换状态
		ELSIF st_IOData.I_CalSignal=1 THEN
			_diCmdState :=19;
		END_IF
		
	22://单元实际液量设定
		_tonDelay(IN:= TRUE,pt:=T#20MS);//保证执行的是最新的一次
		st_IOData.O_ModuleRealVolume := stRunPara.rModuleRealFluVolume	;	
		IF _tonDelay.Q
		THEN	
			IF ABS(st_IOData.O_ModuleRealVolume-st_IOData.O_FluVolumeSet)<0.5 THEN//误差不能超过0.3ml
				stPara.pCtlSignal[12] := TRUE;//
			ELSE
				eERRORID := RudongPump_ERROR.FLT_PumpCal_OverFlow;//误差过大
				_diCmdState := 999;
			END_IF	
			//复位定时器
			_tonDelay(IN:=FALSE);
			_tonCmdTimeout(in:=FALSE);
			_tonTimeout(in:=FALSE);
			_diCmdState := _diCmdState+1;//切换状态
		END_IF
		
	23://等待单元实际液量设定被响应
		_tonCmdTimeout(IN:= stPara.pCtlSignal[12],pt:=T#2S);
		IF NOT stPara.pCtlSignal[12]//
		THEN		
			_tonDelay(IN:=TRUE,PT:= T#50MS);
			IF _tonDelay.Q
			THEN
				_tonTimeout(in:=FALSE);
				_tonDelay(IN:=FALSE);
				_tonCmdTimeout(IN:= FALSE); 
				_diCmdState := _diCmdState+1;//切换状态
			END_IF	
		END_IF	
		IF _tonCmdTimeout.Q
		THEN
			eERRORID := RudongPump_ERROR.FLT_CMD_TIMEOUT;		
			_diCmdState := 999;
		END_IF		
*)
	21://
		IF st_IOData.I_CalSignal=0 THEN
			xComplete := TRUE; 
		ELSE
			_diCmdState :=19;
		END_IF
		
	ELSE
		;	
END_CASE
END_METHOD

METHOD PROTECTED CmdRunAction
VAR_OUTPUT
	xComplete: BOOL;
END_VAR
// return the real actual fault number
IF eERRORID <> RudongPump_ERROR.No_ERROR
THEN
  RETURN;  
END_IF

CASE _diCmdState OF	
	0://传送力值和速度参数	  	
		IF xNeedConfigurePara
		THEN
			_tonDelay(IN:= TRUE,pt:=T#100MS);//保证执行的是最新的一次
			//st_IOData.O_RunModeSet := 2	;//打开定时定量模式
			IF _tonDelay.Q
			THEN	
				//复位定时器
				_tonDelay(IN:=FALSE);
				_tonCmdTimeout(in:=FALSE);
				_tonTimeout(in:=FALSE);
				_diCmdState := _diCmdState+1;//切换状态
			END_IF
			//复位定时器
			_tonDelay(IN:=FALSE);
			_tonCmdTimeout(in:=FALSE);
			_tonTimeout(in:=FALSE);
			_diCmdState := _diCmdState+1;//切换状态
		ELSE//直接启动就好
			//复位定时器
			_tonDelay(IN:=FALSE);
			_tonCmdTimeout(in:=FALSE);
			_tonTimeout(in:=FALSE);
			_diCmdState := 8;//切换状态
		END_IF	
		//检测流量转速是否在0.1rpm - 600rpm
		IF 	rRuntimeSet = 0 
		THEN 
			eERRORID := RudongPump_ERROR.FLT_FLUVOLUM_TIME_PARA;		
			_diCmdState := 999;
		ELSE
			_rSetSpeed := rFluVolumeSet * 60.0 / rSpeedRatio / rRuntimeSet;
			IF _rSetSpeed >= 0.001 AND _rSetSpeed <= 600
			THEN
				;
			ELSE
				eERRORID := RudongPump_ERROR.FLT_FLUVOLUM_TIME_PARA;		
				_diCmdState := 999;
			END_IF
		END_IF				
		
	1://等待定时定量模式被响应
		_tonDelay(IN:=TRUE,PT:= T#50MS);
		IF _tonDelay.Q
		THEN			
			_tonTimeout(in:=FALSE);
			_tonDelay(IN:=FALSE);
			_tonCmdTimeout(IN:= FALSE);   
			_diCmdState := _diCmdState+1;//切换状态
		END_IF	   		
		IF _rxState=999
		THEN
			eERRORID := RudongPump_ERROR.FLT_CMD_TIMEOUT;		
			_diCmdState := 999;
		END_IF		

//发送虚假定量时间		
	2://定量时间设定	
		st_IOData.O_RuntimeSet :=iMaxRunTime-1	;	//保证电机转速不会超
	  SysMemCpy(ADR(_aAddr[7,1]),ADR(st_IOData.O_RuntimeSet),4);
	  _wRuntimeSetTemp := TO_WORD(_aAddr[7,1]);
	  _aAddr[7,1] :=_AADDR[7,2];
	  _aAddr[7,2] :=TO_INT(_wRuntimeSetTemp); 		
		_tonDelay(IN:= TRUE,pt:=T#30MS);//保证执行的是最新的一次
		IF _tonDelay.Q
		THEN	
			_aExecute[7] := TRUE;//启动夹紧控制数据发送	
			//复位定时器
			_tonDelay(IN:=FALSE);
			_tonCmdTimeout(in:=FALSE);
			_tonTimeout(in:=FALSE);
			_diCmdState := _diCmdState+1;//切换状态
		END_IF
	3://等待定量时间设定被响应
		IF NOT _aExecute[7]
		THEN	
			_tonDelay(IN:=TRUE,PT:= T#50MS);
			IF _tonDelay.Q
			THEN				
				_tonTimeout(in:=FALSE);
				_tonDelay(IN:=FALSE);
				_tonCmdTimeout(IN:= FALSE);    
				_diCmdState := _diCmdState+1;//切换状态
			END_IF					
		END_IF	
		IF _rxState=999
		THEN
			eERRORID := RudongPump_ERROR.FLT_CMD_TIMEOUT;		
			_diCmdState := 999;
		END_IF	
		
//传递液量参数		
	4://传送力值和速度参数		
		_tonDelay(IN:= TRUE,pt:=T#30MS);//保证执行的是最新的一次
		st_IOData.O_FluVolumeSet := rFluVolumeSet	;
	  SysMemCpy(ADR(_aAddr[6,1]),ADR(st_IOData.O_FluVolumeSet),4);	
	  _wFluVolumeSetTemp := TO_WORD(_aAddr[6,1]);
	  _aAddr[6,1] := _aAddr[6,2];
	  _aAddr[6,2] := TO_INT(_wFluVolumeSetTemp);	
		IF _tonDelay.Q
		THEN	
		  dwTest1:=	  dwTest1+1;
			_aExecute[6] := TRUE;//启动夹紧控制数据发送	
			//复位定时器
			_tonDelay(IN:=FALSE);
			_tonCmdTimeout(in:=FALSE);
			_tonTimeout(in:=FALSE);
			_diCmdState := _diCmdState+1;//切换状态
		END_IF	  
	5://等待流量设定结束
		IF NOT _aExecute[6]//
		THEN	
			_tonDelay(IN:=TRUE,PT:= T#50MS);
			IF _tonDelay.Q
			THEN					
				_tonTimeout(in:=FALSE);
				_tonDelay(IN:=FALSE);
				_tonCmdTimeout(IN:= FALSE);    
				_diCmdState := _diCmdState+1;//切换状态
			END_IF					
		END_IF	
		IF _rxState=999
		THEN
			eERRORID := RudongPump_ERROR.FLT_CMD_TIMEOUT;		
			_diCmdState := 999;
		END_IF

//传递实际定量时间		
	6://定量时间设定	
		st_IOData.O_RuntimeSet := rRuntimeSet	;	
	  SysMemCpy(ADR(_aAddr[7,1]),ADR(st_IOData.O_RuntimeSet),4);
	  _wRuntimeSetTemp := TO_WORD(_aAddr[7,1]);
	  _aAddr[7,1] := _aAddr[7,2];
	  _aAddr[7,2] := TO_INT(_wRuntimeSetTemp);		
		_tonDelay(IN:= TRUE,pt:=T#25MS);//保证执行的是最新的一次
		IF _tonDelay.Q
		THEN	
			_aExecute[7] := TRUE;//启动夹紧控制数据发送	
			//复位定时器
			_tonDelay(IN:=FALSE);
			_tonCmdTimeout(in:=FALSE);
			_tonTimeout(in:=FALSE);
			_diCmdState := _diCmdState+1;//切换状态
		END_IF
		
	7://等待定量时间设定被响应
		IF NOT _aExecute[7]//
		THEN		
			_tonDelay(IN:=TRUE,PT:= T#50MS);
			IF _tonDelay.Q
			THEN			
				_tonTimeout(in:=FALSE);
				_tonDelay(IN:=FALSE);
				_tonCmdTimeout(IN:= FALSE);    
				_diCmdState := _diCmdState+1;//切换状态
			END_IF				
		END_IF	
		IF _rxState=999
		THEN
			eERRORID := RudongPump_ERROR.FLT_CMD_TIMEOUT;		
			_diCmdState := 999;
		END_IF	
		
	8://方向设定		
		_tonDelay(IN:= ( eCmd = RudongPump_CMD.Cmd_Push OR eCmd = RudongPump_CMD.Cmd_Pull ) ,pt:=T#20MS);//保证执行的是最新的一次
		//IF   eCmd = RudongPump_CMD.Cmd_Push
		//THEN
		//	st_IOData.O_DirectionSet := 1	;			
		//END_IF
		//IF eCmd = RudongPump_CMD.Cmd_Pull 
		//THEN
		//	st_IOData.O_DirectionSet := 0	;			
		//END_IF
		st_IOData.O_DirectionSet:=iDirectionSet;
		IF _tonDelay.Q
		THEN	
			_aExecute[4] := TRUE;//启动夹紧控制数据发送	
			//复位定时器
			_tonDelay(IN:=FALSE);
			_tonCmdTimeout(in:=FALSE);
			_tonTimeout(in:=FALSE);
			_diCmdState := _diCmdState+1;//切换状态
		END_IF
		
	9://等待方向设定被响应
		IF NOT _aExecute[4]//
		THEN		
			_diCmdState := _diCmdState +1; 
			_tonDelay(IN:=FALSE);
			_tonCmdTimeout(in:=FALSE);
			_tonTimeout(in:=FALSE);
		END_IF	
		IF _rxState=999
		THEN
			eERRORID := RudongPump_ERROR.FLT_CMD_TIMEOUT;		
			_diCmdState := 999;
		END_IF	
		
	10://重复次数设定		
		_tonDelay(IN:= TRUE,pt:=T#25MS);//保证执行的是最新的一次
		st_IOData.O_CycleNumber := iCycleNumber	;	
		IF _tonDelay.Q
		THEN	
			_aExecute[9] := TRUE;//启动夹紧控制数据发送	
			//复位定时器
			_tonDelay(IN:=FALSE);
			_tonCmdTimeout(in:=FALSE);
			_tonTimeout(in:=FALSE);
			_diCmdState := _diCmdState+1;//切换状态
		END_IF
		
	11://等待重复次数设定被响应
		IF NOT _aExecute[9]//
		THEN	
			_tonDelay(IN:=TRUE,PT:= T#50MS);
			IF _tonDelay.Q
			THEN	
				_tonTimeout(in:=FALSE);
				_tonDelay(IN:=FALSE);
				_tonCmdTimeout(IN:= FALSE); 
				_diCmdState := _diCmdState+3;//切换状态
			END_IF					
		END_IF	
		IF _rxState=999
		THEN
			eERRORID := RudongPump_ERROR.FLT_CMD_TIMEOUT;		
			_diCmdState := 999;
		END_IF	

//	12://回吸角度		
//		_tonDelay(IN:= TRUE,pt:=T#25MS);//保证执行的是最新的一次
//		st_IOData.O_BackAngle := iBackAngle	;	
//		IF _tonDelay.Q
//		THEN	
//			_aExecute[8] := TRUE;//启动夹紧控制数据发送	
//			//复位定时器
//			_tonDelay(IN:=FALSE);
//			_tonCmdTimeout(in:=FALSE);
//			_tonTimeout(in:=FALSE);
//			_diCmdState := _diCmdState+1;//切换状态
//		END_IF
//		
//	13://等待回吸角度设定响应
//		IF NOT _aExecute[8]//
//		THEN	
//			_tonDelay(IN:=TRUE,PT:= T#50MS);
//			IF _tonDelay.Q
//			THEN	
//				_tonTimeout(in:=FALSE);
//				_tonDelay(IN:=FALSE);
//				_tonCmdTimeout(IN:= FALSE); 
//				_diCmdState :=  _diCmdState+1;//切换状态
//			END_IF					
//		END_IF	
//		IF _rxState=999
//		THEN
//			eERRORID := RudongPump_ERROR.FLT_CMD_TIMEOUT;		
//			_diCmdState := 999;
//		END_IF	
	
		
	14://启动设定		
		_tonDelay(IN:= TRUE ,pt:=T#25MS);//保证执行的是最新的一次	
		st_IOData.O_ControlSet := 1	;					
		IF _tonDelay.Q
		THEN	
			_aExecute[3] := TRUE;//启动夹紧控制数据发送	
			//复位定时器
			_tonDelay(IN:=FALSE);
			_tonCmdTimeout(in:=FALSE);
			_tonTimeout(in:=FALSE);
			_diCmdState := _diCmdState+1;//切换状态
		END_IF
	
	15://等待启动被响应			
		IF  NOT _aExecute[3] THEN
			_tonDelay(IN:= TRUE ,pt:=T#200MS);//等待蠕动泵运行
			IF _tonDelay.Q
			THEN
				_tonDelay(IN:=FALSE);
				_tonCmdTimeout(in:=FALSE);
				_tonTimeout(in:=FALSE);
				_diCmdState := _diCmdState+1;
			END_IF			
		END_IF	
		IF _rxState=999
		THEN
			eERRORID := RudongPump_ERROR.FLT_CMD_TIMEOUT;		
			_diCmdState := 999;
		END_IF			
	16://读取运行状态
		_tonCmdTimeout(in:=FALSE);
		_tonDelay(IN:=TRUE,PT:=T#25MS); 
		_tonTimeout(in:=TRUE,pt:=T#10S);//设置超时时间
    IF  _tonDelay.Q THEN
			_aExecute[16] := TRUE;//触发读取反馈数据 
		  _tonDelay(IN:=FALSE);
			_diCmdState := _diCmdState +1; 	 
    END_IF 		
	17://等待状态响应
		_tonTimeout(in:=TRUE,pt:=T#10S);	  
	  //进行数据刷新  
	  IF NOT _aExecute[16] //等待读取数据完成
	  THEN 
			_tonDelay(IN:= TRUE,pt:=T#40MS);//设置刷新周期	
			IF _tonDelay.Q			 
			THEN
				 _aExecute[16] := FALSE;//触发读取反馈数据 
				 _aRead_VAR.bExecute:=FALSE;
				 _tonDelay(IN:=FALSE);
				 _diCmdState:=16;//回到上一步重新进行状态刷新
			END_IF  
	    SysMemCpy(ADR(st_IOData.I_RunSignal),ADR(_aAddr[16,1]),2);
	    IF st_IOData.I_RunSignal = 0 
	    THEN
				_tonCmdTimeout(in:=FALSE);
				_tonDelay(IN:= FALSE);
				_tonTimeout(in:=FALSE);  
				_diCmdState := 100;
				xComplete := TRUE;
	    END_IF 				
			IF _tonTimeout.Q//旋转动作超时
			THEN
				IF eCmd = RudongPump_CMD.Cmd_Push
				THEN
					eERRORID := RudongPump_ERROR.FLT_PUSH_TIMEOUT;		
				END_IF
				IF eCmd = RudongPump_CMD.Cmd_Pull 
				THEN
					eERRORID := RudongPump_ERROR.FLT_PULL_TIMEOUT;			
				END_IF	
			 _diCmdState := 999;
			END_IF
  	END_IF 
		IF _rxState=999//
			THEN
				eERRORID := eERRORID := RudongPump_ERROR.FLT_CMD_TIMEOUT;
				_diCmdState := 999;
			END_IF
	ELSE
		;	
END_CASE
END_METHOD

ACTION ConnectAction:

//_iChannelIndex := 16;
CASE _iChannelIndex OF 
	1..15:	
		  _aWrite_VAR(
			sIPAddr:= stPara.strSlaveIP, 
			nTCPPort:= stPara.iSlavePort, 
			nUnitID:= stPara.bySlaveID, 
			nQuantity:= _aQuantity[_iChannelIndex], 
			nMBAddr:= _aMBAddr[_iChannelIndex], 
			cbLength:= _aQuantity[_iChannelIndex] * 2, 
			pSrcAddr:= ADR(_aAddr[_iChannelIndex,1]), 
			bExecute:=, 
			tTimeout:= T#3S, 
			bBusy=> , 
			bError=> , 
			nErrId=> );	

	16,17:	      	
		  _aRead_VAR(
			sIPAddr:= stPara.strSlaveIP, 
			nTCPPort:= stPara.iSlavePort, 
			nUnitID:= stPara.bySlaveID, 
			nQuantity:= _aQuantity[_iChannelIndex], 
			nMBAddr:= _aMBAddr[_iChannelIndex], 
			cbLength:= _aQuantity[_iChannelIndex] * 2, 
			pDestAddr:=  ADR(_aAddr[_iChannelIndex,1]), 
			bExecute:= , 
			tTimeout:=T#3S  , 
			bBusy=> , 
			bError=> , 
			nErrId=> , 
			cbRead=> );	
	ELSE
	
	;	
END_CASE	 		

//收发流程管控
CASE _rxState OF 
	0:
    _aWrite_VAR(bExecute:=FALSE);
    _aRead_VAR(bExecute:=FALSE);
	  _iChannelIndex:=0;	
		_rxState := _rxState + 1;		
			
	1:
	  //ACT_GetModbusAdr();
		FOR i := 1 TO 17 BY 1//进行读取指令的轮训
		DO
		 IF _aExecute[i]//检测有控制指令发生
		 THEN
			 _iChannelIndex:=i;
      EXIT;    
			END_IF 
		END_FOR
		IF _iChannelIndex>=16 AND _iChannelIndex<=17//有读取反馈指令
		THEN								
			IF NOT _aRead_VAR.bBusy 
			THEN
				_aRead_VAR(//nMBAddr:= _aMBAddr[_iChannelIndex], 
					          nQuantity:= _aQuantity[_iChannelIndex], 
										nMBAddr:= _aMBAddr[_iChannelIndex], 
										cbLength:= _aQuantity[_iChannelIndex] * 2, 
										pDestAddr:=  ADR(_aAddr[_iChannelIndex,1]), 
                    bExecute := _aExecute[_iChannelIndex]);
				_rxState := _rxState+1;													
			END_IF													
		END_IF			
		IF _iChannelIndex>0 AND _iChannelIndex<16 //有控制触发指令
		THEN		
			IF  NOT _aWrite_VAR.bBusy //AND NOT _aWrite_VAR.bError 
			THEN
				_aWrite_VAR(//nMBAddr:= _aMBAddr[_iChannelIndex],
					          nQuantity:= _aQuantity[_iChannelIndex], 
										nMBAddr:= _aMBAddr[_iChannelIndex], 
										cbLength:= _aQuantity[_iChannelIndex] * 2, 
										pSrcAddr:= ADR(_aAddr[_iChannelIndex,1]), 
                    bExecute := _aExecute[_iChannelIndex]);
				_rxState := _rxState+1;						
			END_IF
		END_IF
		_tonDelay1(in:=FALSE);	
    eMobbusErrorID := 0;		
	2://数据解析		
		_tonDelay1(IN:= TRUE,PT:=T#3S);				
		IF _iChannelIndex>=16
		THEN					
			IF NOT _aRead_VAR.bBusy AND NOT _aRead_VAR.bError//AND NOT _aRead_VAR.bError
			THEN
				_iComNGCount := 0;
				_aExecute[_iChannelIndex] := FALSE;
				_aRead_VAR.bExecute := FALSE;
				_rxState := 0;//等待下次触发
			END_IF
			IF _aRead_VAR.bError
			THEN
				_iComNGCount := _iComNGCount + 1;//错误次数加一
				IF _iComNGCount >= 3//重发多次失败
				THEN
					eMobbusErrorID := _aRead_VAR.nErrId;
					_aRead_VAR.bExecute := FALSE;
					_rxState := 999;//进入错误发生状态
				ELSE
					_tonDelay1(in:=FALSE);
					_aRead_VAR.bExecute:= FALSE;
					_rxState := _rxState + 1;
				END_IF						
			END_IF			
		END_IF				
		IF _iChannelIndex>=1 AND _iChannelIndex<=15		
		THEN	
			IF NOT _aWrite_VAR.bBusy AND NOT _aWrite_VAR.bError//AND NOT _aWrite_VAR.bError
			THEN
				_iComNGCount := 0;
				_aExecute[_iChannelIndex] := FALSE;
				_aWrite_VAR.bExecute := FALSE;
				_rxState := 0;//等待下次触发
			END_IF
			IF _aWrite_VAR.bError
			THEN
				_iComNGCount := _iComNGCount + 1;//错误次数加一
				IF _iComNGCount >= 3//重发多次失败
				THEN
					eMobbusErrorID := _aWrite_VAR.nErrId;
					_aWrite_VAR.bExecute := FALSE;
					_rxState := 999;//进入错误发生状态
				ELSE
					_tonDelay1(in:=FALSE);
					_aWrite_VAR.bExecute:= FALSE;
					_rxState := _rxState + 1;
				END_IF					
			END_IF				
		END_IF	
    IF _tonDelay1.Q//超时
		THEN
			_rxState:= 999;					
		END_IF				
	3://delay
		_tonDelay1(in:=TRUE,PT:=T#60MS);
		_aWrite_VAR(bExecute:=FALSE);
    _aRead_VAR(bExecute:=FALSE);
		IF _tonDelay1.Q
		THEN
			_rxState := 0;			
			_tonDelay1(in:=FALSE);	
    END_IF	
	999://错误状态，等待复位发生
		IF _fResetCheck.Q
		THEN
			FOR i:= 1 TO 17 DO
				_aExecute[i] := FALSE;				
			END_FOR
		  _iChannelIndex:=0;
			_aWrite_VAR.bExecute:=FALSE;
			_aRead_VAR.bExecute:=FALSE;			
			_iComNGCount := 0;//
			_rxState := 0;//重新开始			
		END_IF
	ELSE
		;
END_CASE
END_ACTION

METHOD PROTECTED CyclicAction
VAR_INPUT
END_VAR
VAR_OUTPUT
	xComplete: BOOL;
END_VAR
VAR	
END_VAR
IF xAbort=0 THEN
    IF xFirstInvocation THEN
    (*
    * Staring
    * for then first (!) invocaion,
    * sample then input variables
    *)			
    _diCmdState:= 0;
		_iNGCount := 0;
		_iActRunNumber := 0;
		xFirstInvocation:=0;			
    END_IF    
    REPEAT 				
		  (**************************检查是否有硬件报错(检测总线是否报错)**********************************) 
			IF _xConnectError
			THEN
				eERRORID := RudongPump_ERROR.FLT_CONNECT;//子站通讯报警
			END_IF
//检测参数是否配置正确			
			IF ( stPara.iType <> 1 AND stPara.iType <> 2 )//只能是modbus模式	 
			THEN
				eERRORID := RudongPump_ERROR.FLT_PARA;//参数配置错误
			END_IF
	
			//检测停止指令是否发生
			_rStopCmdTrig(CLK:= NOT xEStop OR (stDeviceOpe.xStop_Hmi AND NOT xAutoMode AND NOT xDeviceRunning) OR (stDeviceOpe.xStop_Auto AND (xAutoMode OR xDeviceRunning))
													OR (stDeviceOpe.xFullSpeedStop_Hmi AND NOT xAutoMode AND NOT xDeviceRunning) OR (stDeviceOpe.xFullSpeedStop_Auto AND (xAutoMode OR xDeviceRunning)));		
		  IF _rStopCmdTrig.Q//检测到停止指令
			THEN
				_diCmdState := 0;
				eCmd := RudongPump_CMD.Cmd_Stop;
				_tonCmdTimeout(in:=FALSE);
				_tonDelay(IN:= FALSE);
				_tonTimeout(in:=FALSE);
				FOR i:=1 TO 17 BY 1 
				DO 
					_aExecute[i] := FALSE;			
				END_FOR
				_diCmdState := 0;
			END_IF			
			//检测是否有Modbus指令运行中	
			_xCheckModbusRun := FALSE;
			_xBusy:=_aWrite_VAR.bBusy OR _aRead_VAR.bBusy;
			_xCheckModbusRun := _xBusy;	
			ACT_PumpPar();//检查参数
	
			//检测是否有Modbus报错	
			_xError:=_aWrite_VAR.berror OR _aRead_VAR.berror;			
			
			CASE eCmd OF//判断指令类型
				RudongPump_CMD.Cmd_Pull,RudongPump_CMD.Cmd_Push://执行夹爪指令(夹紧和松开指令)
					CmdRunAction(xComplete=> xComplete);	
							
				RudongPump_CMD.Cmd_Stop,RudongPump_CMD.Cmd_FullSpeedStop://执行过程中等待停止指令(分为运行停止和全速停止)
					mCmdStopAction(xComplete=> xComplete);
					
				RudongPump_CMD.Cmd_Configure://(用于配置参数)
					mCmdConfigureAction(xComplete=> xComplete);
					
				RudongPump_CMD.Cmd_FullSpeedPush,RudongPump_CMD.Cmd_FullSpeedPull://全速启动控制（用于清洗和充满试管）
					mCmdFullSpeedStartAction(xComplete=> xComplete);
					
				RudongPump_CMD.Cmd_CalPump:
					CmdPumpCal(xComplete=> xComplete);

				RudongPump_CMD.Cmd_CalReset:
					CmdCalReset(xComplete=> xComplete);		

				RudongPump_CMD.Cmd_CalParWrite:
					CmdCalParWrite(xComplete=> xComplete);		
				ELSE
					;	
				END_CASE		   
      UNTIL (TRUE)
	END_REPEAT
END_IF

IF xAbort OR xComplete OR eERRORID<>RudongPump_ERROR.No_ERROR THEN    
    (*
    * Cleaning
    * => free as much allocated resources as possible
    *)    
    tOperationTimer(IN:=0);
END_IF
END_METHOD

METHOD PRIVATE FINAL HandleAbortedState
VAR_INPUT
END_VAR
VAR_OUTPUT
	xAgain: BOOL;
END_VAR
VAR
	xComplete: BOOL;
END_VAR
IF xAborted AND xResetRequest THEN
    eState:=STATE.RESETING;
    xAgain:=1;
ELSE
    xBusy:=0;
    xAborted:=1;
    //xResetRequest:=(xExecute=0);
    xAgain:=0;(* !!! *)
END_IF
END_METHOD

METHOD PRIVATE FINAL HandleAbortingState
VAR_INPUT
END_VAR
VAR_OUTPUT
	xAgain: BOOL;
END_VAR
VAR
	xComplete: BOOL;
END_VAR
AbortAction(xComplete=> xComplete, eERRORID=> eERRORID);

IF eERRORID<>RudongPump_ERROR.No_ERROR THEN
    eState:=STATE.INERROR;
    xAgain:=1;
ELSIF xComplete THEN
    eState:=STATE.ABORTED;
    xAgain:=1;
END_IF
END_METHOD

METHOD PRIVATE FINAL HandleDoneState
VAR_INPUT
END_VAR
VAR_OUTPUT
	xAgain: BOOL;
END_VAR
//在运行过程中要是切换模式，再运行完成之后，检测到模式的切换，就需要回到初始位置，进行下一次执行准备
IF _xDone AND ((xExecute=0) OR ( _xModeChange AND NOT _xAutoOpe)  OR ( NOT xAutoMode AND NOT xDeviceRunning AND ( NOT _xAutoOpe OR _xHMIOpe))) THEN
	eState:=STATE.RESETING;
	xAgain:=1;
ELSE
	xBusy:=0;
	_xDone:=1;
	xAgain:=0;(* !!! *)
END_IF
END_METHOD

METHOD PRIVATE FINAL HandleDormantState
VAR_INPUT
END_VAR
VAR_OUTPUT
	xAgain: BOOL;
END_VAR
IF xExecute THEN
    xBusy:=1;
    eState:=STATE.EXECUTING;
    xAgain:=1;
END_IF
//下面两个报警一旦报警就需要发生
IF _xConnectError 
THEN//出现这个进行报警
	eERRORID := RudongPump_ERROR.FLT_CONNECT;//子站通讯报警
END_IF

IF _fResetCheck.Q//清空报警
THEN
	eERRORID := RudongPump_ERROR.No_ERROR;
END_IF
IF  xAutoMode OR xDeviceRunning THEN
	xAutomodeFlag:=TRUE;
ELSE
	xAutomodeFlag:=FALSE;
END_IF


IF eErrorID = RudongPump_ERROR.NO_ERROR 
THEN
	IF   xRunILC   THEN
		FOR k:=1 TO 5 BY 1 DO
			//PULL
			_rOperaTrig[k](CLK:=xRunILC AND (stDeviceOpe.xPull_Hmi[k] AND NOT xAutomodeFlag) OR (stDeviceOpe.xPull_Auto[k] AND xAutomodeFlag));
			IF _rOperaTrig[k].Q //
			THEN
				rFluVolumeSet	:=stRunPara.rPullFluVolume[k];
				rRuntimeSet		:=stRunPara.rPullRuntime[k];
				iCycleNumber	:=stRunPara.iPullCycleNumber[k];
				iBackAngle		:=stRunPara.iPullBackAngle[k];
				eCmd 			:= RudongPump_CMD.Cmd_Pull;
				xExecute		:= TRUE;
			END_IF		
			//PUSH
			_rOperaTrig[k+5](CLK:=xRunILC AND (stDeviceOpe.xPush_Hmi[k] AND NOT xAutomodeFlag) OR (stDeviceOpe.xPush_Auto[k] AND xAutomodeFlag));
			IF _rOperaTrig[k+5].Q 
			THEN
				rFluVolumeSet	:=stRunPara.rPushFluVolume[k];  
				rRuntimeSet		:=stRunPara.rPushRuntime[k];    
				iCycleNumber	:=stRunPara.iPushCycleNumber[k];
				iBackAngle		:=stRunPara.iPushBackAngle[k];
				eCmd 			:= RudongPump_CMD.Cmd_Push;
				xExecute 		:= TRUE;
			END_IF				
		END_FOR
		//STOP
		 IF stDeviceOpe.xStop_Hmi OR stDeviceOpe.xStop_Auto OR  NOT xEStop     THEN
				eCmd := RudongPump_CMD.Cmd_Stop;
				xExecute := TRUE;
		 END_IF
		//FullSpeedPull
		IF (stDeviceOpe.xFullSpeedPull_Hmi AND  NOT xAutomodeFlag) OR (stDeviceOpe.xFullSpeedPull_Auto AND  xAutomodeFlag) THEN
			eCmd := RudongPump_CMD.Cmd_FullSpeedPull;
			xExecute := TRUE;
		END_IF
		//FullSpeedPush
		IF (stDeviceOpe.xFullSpeedPush_Hmi AND NOT xAutomodeFlag ) OR (stDeviceOpe.xFullSpeedPush_Auto AND xAutomodeFlag) THEN	
			eCmd := RudongPump_CMD.Cmd_FullSpeedPush;
			xExecute := TRUE;
		END_IF
		//FullSpeedStop
		 IF (stDeviceOpe.xFullSpeedStop_Hmi AND NOT xAutomodeFlag) OR (stDeviceOpe.xFullSpeedStop_Auto AND xAutomodeFlag) THEN	
			eCmd := RudongPump_CMD.Cmd_FullSpeedStop;
			xExecute := TRUE;
		END_IF
		//Configure
		IF (stDeviceOpe.xConfigure_Hmi AND NOT xAutomodeFlag) OR (stDeviceOpe.xConfigure_Auto AND xAutomodeFlag) THEN	
			eCmd := RudongPump_CMD.Cmd_Configure;
			xExecute := TRUE;
		END_IF
		
	END_IF		
		//校准
		IF stDeviceOpe.xPumpCal_Hmi OR stDeviceOpe.xPumpCal_Auto THEN
				rFluVolumeSet		:=stRunPara.rCalFluVolume;
				rRuntimeSet			:=stRunPara.rCalTime;
				iCycleNumber		:=stRunPara.rCalNum;	
				iModuleAdress		:=stRunPara.iModuleAdress;
				iModuleSpeed		:=stRunPara.rCalFluVolume/stRunPara.rCalTime;   //stRunPara.rModuleSpeed;		
				eCmd 				:= RudongPump_CMD.Cmd_CalPump;
				xExecute 			:= TRUE;		
		END_IF
		
		//复位校准系数为初始值
		IF stDeviceOpe.xResetCalcoeffCal_Hmi THEN	
			eCmd 				:= RudongPump_CMD.Cmd_CalReset;
			xExecute 			:= TRUE;		
		END_IF
	
		//校准参数写入
		IF stDeviceOpe.xCalParWrite_Hmi OR stDeviceOpe.xCalParWrite_Auto THEN	
			eCmd 								:= RudongPump_CMD.Cmd_CalParWrite;
			iModuleRealVolume		:=stRunPara.rModuleRealFluVolume;					
			xExecute 						:= TRUE;		
		END_IF	
			
END_IF
END_METHOD

METHOD PRIVATE FINAL  HandleErrorState
VAR_INPUT
END_VAR
VAR_OUTPUT
	xAgain: BOOL;
END_VAR
IF xRudongPump_ERROR AND  (xResetRequest OR NOT xExecute) THEN
    eState:=STATE.RESETING;
    xAgain:=1;
ELSE
    xBusy:=0;
    xRudongPump_ERROR:=1;    
    xAgain:=0;(* !!! *)
END_IF
END_METHOD

METHOD PRIVATE FINAL HandleExecutingState
VAR_INPUT
END_VAR
VAR_OUTPUT
	xAgain: BOOL;
END_VAR
VAR
	xComplete: BOOL;
END_VAR
IF xAbort=0 THEN   
    CyclicAction(xComplete=> xComplete);
END_IF

IF eERRORID<>RudongPump_ERROR.No_ERROR THEN
    eState:=STATE.INERROR;
    xAgain:=1;
ELSIF xAbort THEN
    eState:=STATE.ABORTING;
    xAgain:=1;
ELSIF xComplete THEN
    eState:=STATE.DONE;
    xAgain:=1;
END_IF
END_METHOD

METHOD PRIVATE FINAL HandleResettingState
VAR_INPUT
END_VAR
VAR_OUTPUT
	xAgain: BOOL;
END_VAR
VAR
	xComplete: BOOL;
END_VAR
ResetAction(xComplete=> xComplete);

IF xComplete THEN
	xExecute:=0;//清除输入指令 
    xBusy:=0;
    _xDone:=0;
    xRudongPump_ERROR:=0;
    xAborted:=0;
    eERRORID:=RudongPump_ERROR.No_ERROR;
    eState:=STATE.DORMANT;
    xFirstInvocation:=1;
    xAgain:=0;(* !!! *)
END_IF
END_METHOD

METHOD JudgePar : RudongPump_ERROR
VAR_OUTPUT
	eERRORID: RudongPump_ERROR;(*错误码*)
END_VAR
END_METHOD

METHOD PROTECTED mCmdConfigureAction
VAR_OUTPUT
	xComplete: BOOL;
END_VAR
VAR
END_VAR
// return the real actual fault number
IF eERRORID <> RudongPump_ERROR.No_ERROR
THEN
  RETURN;  
END_IF

CASE _diCmdState OF
	0://使能失效操作	
			//st_IOData.O_PumpType := stRunPara.iPumpTypeSet;
			_tonDelay(IN:=TRUE,PT:=T#25MS);
			IF _tonDelay.Q//等待指令响应
			THEN
				_aExecute[1] := TRUE;//触发运行指令	
				//复位定时器
				_tonTimeout(in:=FALSE);
				_tonDelay(IN:=FALSE);
				_tonCmdTimeout(IN:= FALSE);    
				_diCmdState := _diCmdState+1;//切换状态
			END_IF	  		

	1://等待使能失效被响应	
		IF NOT _aExecute[1]
		THEN
			_tonDelay(IN:=TRUE,PT:= T#50MS);
			IF _tonDelay.Q
			THEN			
				_tonTimeout(in:=FALSE);
				_tonDelay(IN:=FALSE);
				_tonCmdTimeout(IN:= FALSE);    
				_diCmdState := _diCmdState+1;//切换状态
			END_IF			
		END_IF	
		IF _rxState=999//指令超时报错
		THEN
			eERRORID := RudongPump_ERROR.FLT_CMD_TIMEOUT;	
			diStepOld:=	_diCmdState;	
			_diCmdState := 999;
		END_IF	
	2://设置软管类型		
		//st_IOData.O_HosePipeType := stRunPara.iHosePipeTypeSet;
		_tonDelay(IN:=TRUE,PT:=T#25MS);
		IF _tonDelay.Q//等待指令响应
		THEN
			_aExecute[2] := TRUE;//触发运行指令	
			//复位定时器
			_tonTimeout(in:=FALSE);
			_tonDelay(IN:=FALSE);
			_tonCmdTimeout(IN:= FALSE);    
			_diCmdState := _diCmdState+1;//切换状态
		END_IF	
	3://等待使能失效被响应	
		IF NOT _aExecute[2]
		THEN
			_tonCmdTimeout(in:=FALSE);
			_tonDelay(IN:= FALSE);
			_tonTimeout(in:=FALSE);  
			_diCmdState := 100;
			 xComplete := 1;
		END_IF	
		IF _rxState=999//指令超时报错
		THEN
			eERRORID := RudongPump_ERROR.FLT_CMD_TIMEOUT;
			diStepOld:=	_diCmdState;		
			_diCmdState := 999;
		END_IF	 
	ELSE
		;
END_CASE
END_METHOD

METHOD PROTECTED mCmdFullSpeedStartAction
VAR_OUTPUT
	xComplete: BOOL;
END_VAR
VAR
END_VAR
// return the real actual fault number
IF eERRORID <> RudongPump_ERROR.No_ERROR
THEN
  RETURN;  
END_IF

CASE _diCmdState OF
	0://方向设定		
		_tonDelay(IN:= ( eCmd = RudongPump_CMD.Cmd_FullSpeedPush OR eCmd = RudongPump_CMD.Cmd_FullSpeedPull ) ,pt:=T#30MS);//保证执行的是最新的一次
		//IF eCmd = RudongPump_CMD.Cmd_FullSpeedPush
		//THEN
		//	st_IOData.O_DirectionSet := 1	;			
		//END_IF
		//IF eCmd = RudongPump_CMD.Cmd_FullSpeedPull 
		//THEN
		//	st_IOData.O_DirectionSet := 0	;			
		//END_IF
		st_IOData.O_DirectionSet :=iDirectionSet;
		IF _tonDelay.Q
		THEN	
			_aExecute[4] := TRUE;//启动夹紧控制数据发送	
			//复位定时器
			_tonDelay(IN:=FALSE);
			_tonCmdTimeout(in:=FALSE);
			_tonTimeout(in:=FALSE);
			_diCmdState := _diCmdState+1;//切换状态
		END_IF
			
	1://等待方向设定被响应
		IF NOT _aExecute[4]//
		THEN		
			_tonDelay(IN:=TRUE,PT:= T#10MS);
			IF _tonDelay.Q
			THEN			
				_tonTimeout(in:=FALSE);
				_tonDelay(IN:=FALSE);
				_tonCmdTimeout(IN:= FALSE);    
				_diCmdState := _diCmdState+1;//切换状态
			END_IF	
		END_IF	
		IF _rxState=999
		THEN
			eERRORID := RudongPump_ERROR.FLT_CMD_TIMEOUT;		
			_diCmdState := 999;
		END_IF	
	2://使能失效操作		     
		st_IOData.O_FullSpeedControl := 1;		
		_tonDelay(IN:=TRUE,PT:=T#25MS);
		IF _tonDelay.Q//等待指令响应
		THEN
			_aExecute[5] := TRUE;//触发运行指令	
			//复位定时器
			_tonTimeout(in:=FALSE);
			_tonDelay(IN:=FALSE);
			_tonCmdTimeout(IN:= FALSE);    
			_diCmdState := _diCmdState+1;//切换状态
		END_IF
	3://等待使能失效被响应	
		IF NOT _aExecute[5]
		THEN
			_tonCmdTimeout(in:=FALSE);
			_tonDelay(IN:= FALSE);
			_tonTimeout(in:=FALSE);  
			_diCmdState :=_diCmdState+1;
		END_IF	
		IF _rxState=999//指令超时报错
		THEN
			eERRORID := RudongPump_ERROR.FLT_CMD_TIMEOUT;		
			_diCmdState := 999;
		END_IF	

	4://读取运行状态
		_tonCmdTimeout(in:=FALSE);
		_tonDelay(IN:=TRUE,PT:=T#25MS); 
    IF  _tonDelay.Q THEN
			_aExecute[16] := TRUE;//触发读取反馈数据 
		  _tonDelay(IN:=FALSE);
			_diCmdState := _diCmdState +1; 	 
    END_IF 	
		
	5://等待状态响应
		_tonTimeout(in:=TRUE,pt:=T#10S);	  
	  //进行数据刷新  
	  IF NOT _aExecute[16] //等待读取数据完成
	  THEN 
			_tonDelay(IN:= TRUE,pt:=T#40MS);//设置刷新周期	
			IF _tonDelay.Q			 
			THEN
				 _aExecute[16] := FALSE;//触发读取反馈数据 
				 _aRead_VAR.bExecute:=FALSE;
				 _tonDelay(IN:=FALSE);
				 _diCmdState:=_diCmdState -1;//回到上一步重新进行状态刷新
			END_IF  
	    SysMemCpy(ADR(st_IOData.I_RunSignal),ADR(_aAddr[16,1]),2);
	    IF st_IOData.I_RunSignal = 1 
	    THEN
				_tonCmdTimeout(in:=FALSE);
				_tonDelay(IN:= FALSE);
				_tonTimeout(in:=FALSE);  
				_diCmdState := 100;
				xComplete := TRUE;
	    END_IF 				
			IF _tonTimeout.Q//旋转动作超时
			THEN
				IF eCmd = RudongPump_CMD.Cmd_Push
				THEN
					eERRORID := RudongPump_ERROR.FLT_PUSH_TIMEOUT;		
				END_IF
				IF eCmd = RudongPump_CMD.Cmd_Pull 
				THEN
					eERRORID := RudongPump_ERROR.FLT_PULL_TIMEOUT;			
				END_IF	
			 _diCmdState := 999;
			END_IF
  	END_IF 
		IF _rxState=999//
			THEN
				eERRORID := eERRORID := RudongPump_ERROR.FLT_CMD_TIMEOUT;
				_diCmdState := 999;
			END_IF	
	ELSE
		;
END_CASE
END_METHOD

METHOD PROTECTED mCmdStopAction
VAR_OUTPUT
	xComplete: BOOL;
END_VAR
VAR
END_VAR
// return the real actual fault number
IF eERRORID <> RudongPump_ERROR.No_ERROR
THEN
  RETURN;  
END_IF

CASE _diCmdState OF
	0://使能失效操作
		st_IOData.O_ControlSet := 0;
		st_IOData.O_FullSpeedControl := 0;		  
		_tonDelay(IN:=TRUE,PT:=T#400MS);
		IF _tonDelay.Q//等待指令响应
		THEN
			IF eCmd = RudongPump_CMD.Cmd_Stop
			THEN
				_aExecute[3] := TRUE;//触发运行指令	
			END_IF
			IF eCmd = RudongPump_CMD.Cmd_FullSpeedStop
			THEN
				_aExecute[5] := TRUE;//触发运行指令	
			END_IF
			//复位定时器
			_tonTimeout(in:=FALSE);
			_tonDelay(IN:=FALSE);
			_tonCmdTimeout(IN:= FALSE);    
			_diCmdState := _diCmdState+1;//切换状态
		END_IF			

	1://等待使能失效被响应	
		IF NOT _aExecute[3] AND  NOT _aExecute[5]
		THEN
			_tonCmdTimeout(in:=FALSE);
			_diCmdState := _diCmdState +1; 
		END_IF	
		IF _rxState=999//指令超时报错
		THEN
			eERRORID := RudongPump_ERROR.FLT_CMD_TIMEOUT;		
			_diCmdState := 999;
		END_IF	
  2://延时100ms错开信号
		_tonDelay(IN:= TRUE,pt:=T#100MS);//设置刷新周期
		IF _tonDelay.Q
		THEN			
			_diCmdState := _diCmdState + 1;
		END_IF
	3://读取运行状态
		_tonCmdTimeout(in:=FALSE);	
		_tonTimeout(in:=TRUE,pt:=T#10S);//设置超时时间 	
		_aExecute[16] := TRUE;//触发读取反馈数据 
		_tonDelay(IN:=FALSE);
		_diCmdState := _diCmdState +1;   
	4://等待状态响应
		_tonTimeout(in:=TRUE,pt:=T#10S);	  
	  //进行数据刷新  
	  IF NOT _aExecute[16] //等待读取数据完成
	  THEN 
			_tonDelay(IN:= TRUE,pt:=T#40MS);//设置刷新周期	
			IF _tonDelay.Q			 
			THEN
				 _aExecute[16] := FALSE;//触发读取反馈数据 
				 _aRead_VAR.bExecute:=FALSE;
				 _tonDelay(IN:=FALSE);
				 _diCmdState:=_diCmdState -1;//回到上一步重新进行状态刷新
			END_IF  
	    SysMemCpy(ADR(st_IOData.I_RunSignal),ADR(_aAddr[16,1]),2);
	    IF st_IOData.I_RunSignal = 0 
	    THEN
				_tonCmdTimeout(in:=FALSE);
				_tonDelay(IN:= FALSE);
				_tonTimeout(in:=FALSE);  
				_diCmdState := 100;
				xComplete := TRUE;
	    END_IF 				
			IF _tonTimeout.Q//旋转动作超时
			THEN
				IF eCmd = RudongPump_CMD.Cmd_Push
				THEN
					eERRORID := RudongPump_ERROR.FLT_PUSH_TIMEOUT;		
				END_IF
				IF eCmd = RudongPump_CMD.Cmd_Pull 
				THEN
					eERRORID := RudongPump_ERROR.FLT_PULL_TIMEOUT;			
				END_IF	
			 _diCmdState := 999;
			END_IF
  	END_IF 
		IF _rxState=999//
			THEN
				eERRORID := eERRORID := RudongPump_ERROR.FLT_CMD_TIMEOUT;
				_diCmdState := 999;
			END_IF 		
	ELSE
		;
END_CASE
END_METHOD

METHOD PROTECTED ResetAction
VAR_INPUT
END_VAR
VAR_OUTPUT
	xComplete: BOOL;
END_VAR
(*
* Cleaning
* => free all allocated resources
* => reinitialize instance variables
*)
tOperationTimer(IN:=0);
tInvocationTimer(IN:=0);

// init command state
_diCmdState := 0;
_tonCmdTimeout(in:=FALSE);
_tonDelay(IN:= FALSE);
_tonTimeout(in:=FALSE);
_xModeChange := FALSE;
_rStopCmdTrig(CLK:=FALSE);
_iNGCount := 0;

//清除触发标志位
FOR i:=1 TO 17 BY 1 
DO 
	_aExecute[i] := FALSE;			
END_FOR
_aWrite_VAR.bExecute:=FALSE;
_aRead_VAR.bExecute:=FALSE;	
//清除触发状态
FOR k:=1 TO 15 BY 1 DO
	_rOperaTrig[k](CLK:=FALSE);
END_FOR	
	
stDeviceOpe.xConfigure_Auto:= stDeviceOpe.xConfigure_Hmi:= FALSE;
stDeviceOpe.xStop_Auto:= stDeviceOpe.xStop_Hmi:= FALSE;
stDeviceOpe.xFullSpeedPull_Auto:= stDeviceOpe.xFullSpeedPull_Hmi:= FALSE;
stDeviceOpe.xFullSpeedPush_Auto:= stDeviceOpe.xFullSpeedPush_Hmi:= FALSE;
stDeviceOpe.xFullSpeedStop_Auto:= stDeviceOpe.xFullSpeedStop_Hmi:= FALSE;
FOR k:=1 TO 5 DO
	stDeviceOpe.xPull_Auto[k]:= stDeviceOpe.xPull_Hmi[k] := FALSE;
	stDeviceOpe.xPush_Auto[k]:= stDeviceOpe.xPush_Hmi[k] := FALSE;
END_FOR

stDeviceOpe.xPumpCal_Auto:=stDeviceOpe.xPumpCal_Hmi:=FALSE;
stDeviceOpe.xCalParWrite_Auto:=stDeviceOpe.xCalParWrite_Hmi:=FALSE;
stDeviceOpe.xResetCalcoeffCal_Hmi:=FALSE;
st_IOData.O_ModuleStart := 0	;
xResetRequest:=FALSE;
//复位完成
xComplete:=1;
END_METHOD

END_FUNCTION_BLOCK

// ---- POUs/003_FB/100_test/FB_GetTime.TcPOU
FUNCTION_BLOCK FB_GetTime
VAR_INPUT
	i_b_start:			BOOL;
	i_b_withoutHs:		BOOL;
END_VAR
VAR_OUTPUT
	o_b_ok:				BOOL;
	o_b_err:				BOOL;
	o_udi_ErrId:		UDINT;
	o_DateAndTime:		tDateAndTime;
END_VAR
VAR
	l_b_repeat:			BOOL;
	l_b_repeatOk:		BOOL;
	l_i_step:			INT := 100;
	l_fb_read:			ADSREAD;
END_VAR


(* @END_DECLARATION := '0' *)
REPEAT
	l_b_repeat := FALSE;
	CASE l_i_step OF

		100: (* initial step *)
			IF i_b_start THEN
				l_i_step := 200;
				l_b_repeat := TRUE;
				l_b_repeatOk := FALSE;
			END_IF;

		200:	(* read *)
			l_fb_read(	NETID := '',
							PORT := 10000,
							IDXGRP := 400,
							IDXOFFS := 1,
							LEN := 16,
							DESTADDR := ADR(o_DateAndTime),
							READ := TRUE,
							TMOUT := t#2s);
			IF l_fb_read.busy THEN
				l_b_repeatOk := TRUE;
			END_IF
			IF NOT l_fb_read.busy AND NOT l_fb_read.err THEN
				(* fertig und "no error" *)
				o_b_ok := TRUE;
				o_udi_ErrId := l_fb_read.ErrId;
				l_fb_read(read := FALSE);
				l_i_step := 500;
				l_b_repeat := l_b_repeatOk;
			END_IF;
			IF l_fb_read.err THEN
				(* "error" *)
				o_b_err:=TRUE;
				o_udi_ErrId := l_fb_read.ErrId;
				l_fb_read(read := FALSE);
				l_i_step := 500;
			END_IF;

		500:	(* back *)
			IF NOT i_b_start OR i_b_withoutHs THEN
				l_i_step := 100;
				o_b_ok := FALSE;
				o_b_err := FALSE;
				l_b_repeat := TRUE;
			END_IF;
	END_CASE;
UNTIL l_b_repeat = FALSE
END_REPEAT;

END_FUNCTION_BLOCK

// ---- POUs/003_FB/53_RudongPump/09_PeristalticPumpFB/FB_RuDongPump_ModbusTCP.TcPOU
///{attribute 'hide'}
FUNCTION_BLOCK FB_RuDongPump_ModbusTCP
VAR_INPUT
	xExecute: BOOL;
	xAbort: BOOL;
	///匹配复位按钮 
	xResetRequest: BOOL;
	///蠕动泵运行条件
	xRunILC: BOOL;
	///[ms],1 => no invocation time limit
	dwTimeLimit: DWORD := 1;
	///[ms],0 => no executing time limit
	dwTimeOut: DWORD;
	stPara: RudongPump_Sys_Para_1;
	///是否需要配置参数(默认是需要进行参数配置的)	
	xNeedConfigurePara: BOOL := TRUE;
	///运行参数	
	stRunPara: RudongPump_RunData;
	///0:mannal 1:auto
	xAutoMode: BOOL;
	///初始化过程中
	xIniting: BOOL;
	///工站单循环中
	xDeviceRunning: BOOL;
	///根据泵头软管型号不同有变化
	rSpeedRatio: REAL := 2.733;
	sHmiError: STRING;
	xEStop: BOOL;
	///操作按钮
	stDeviceOpe: RudongPump_Ope_1;
END_VAR
VAR_OUTPUT
	///完成条件满足
	xDone: BOOL;
	///动作正在执行
	xBusy: BOOL;
	///报警中
	xError: BOOL;
	///指令被打断
	xAborted: BOOL;
	///蠕动泵运行中
	xRunning: BOOL;
	///错误条件满足
	xRudongPump_ERROR: BOOL;
	///错误码
	eERRORID: RudongPump_ERROR;
	xRdyCmd: BOOL;
	///最大运行时间,单位s
	iMaxRunTime: REAL;
	///最小运行时间,单位s
	iMinRunTime: REAL;
END_VAR
VAR
	{attribute 'hide' := ''}
	stModbusAddress: RuDongPump_ModbusAddress;
	{attribute 'hide' := ''}
	_pDataControl: POINTER TO BYTE;
	{attribute 'hide' := ''}
	eState: STATE;
	{attribute 'hide' := ''}
	_fbModbusTCP: FB_ModbusTCP;
	{attribute 'hide' := ''}
	_xDone: BOOL;
	///指令控制	
	{attribute 'hide' := ''}
	eCmd: RudongPump_CMD;
	{attribute 'hide' := ''}
	xFirstInvocation: BOOL := TRUE;
	{attribute 'hide' := ''}
	xTimeOut: BOOL;
	{attribute 'hide' := ''}
	xTimeLimit: BOOL;
	{attribute 'hide' := ''}
	tInvocationTimer: TON;
	tOperationTimer: TON;
	///液量设定 0.0-99999.0 mL(0.1ml)
	{attribute 'hide' := ''}
	rFluVolumeSet: REAL;
	///运行时间设定 0.1-9999s(0.1s)
	{attribute 'hide' := ''}
	rRuntimeSet: REAL;
	///重复次数
	{attribute 'hide' := ''}
	iCycleNumber: INT;
	///灌装单元地址
	{attribute 'hide' := ''}
	iModuleAdress: INT;
	///灌装单元速度
	{attribute 'hide' := ''}
	iModuleSpeed: REAL;
	///灌装实际液量	
	{attribute 'hide' := ''}
	iModuleRealVolume: REAL;
	{attribute 'hide' := ''}
	_cmdStop: BOOL;
	{attribute 'hide' := ''}
	_tonTimeout: TON;
	_tonCmdTimeout: TON;
	/// command execution
	{attribute 'hide' := ''}
	_CmdExe: BOOL;
	/// detect rising edge of command execution
	{attribute 'hide' := ''}
	_rTrigCmdExe: R_TRIG;
	{attribute 'hide' := ''}
	_rTrigCmdOrg: R_TRIG;
	{attribute 'hide' := ''}
	_diCmdState: DINT;
	/// detect FltQuit rising edge
	{attribute 'hide' := ''}
	_rTrigFltReset: R_TRIG;
	{attribute 'hide' := ''}
	_tonDelay: TON;
	///	_fbGET_MODBUSTCP_SLAVE_DIAGNOSE_RTU : SysHC_ModbusRtuSlaveDiagnose;//modbusTCP子站诊断函数
	///_fbGET_MODBUSTCP_SLAVE_DIAGNOSE_TCP : GET_MODBUSTCP_SLAVE_DIAGNOSE;//modbusTCP子站诊断函数
	{attribute 'hide' := ''}
	_iConnectState: INT := 0;
	{attribute 'hide' := ''}
	_connectTon: TON;
	{attribute 'hide' := ''}
	_xConnectError: BOOL;
	{attribute 'hide' := ''}
	_fResetCheck: F_TRIG;
	{attribute 'hide' := ''}
	_rManual: R_TRIG;
	{attribute 'hide' := ''}
	_fManual: F_TRIG;
	{attribute 'hide' := ''}
	_xModeChange: BOOL;
	{attribute 'hide' := ''}
	i: INT;
	///状态读取计时定时器
	{attribute 'hide' := ''}
	_tonPulse: TON;
	///检测modbus是否处理总
	{attribute 'hide' := ''}
	_xCheckModbusRun: BOOL;
	///需要匹配参数是OK的
	{attribute 'hide' := ''}
	_xConfigureParaOK: BOOL;
	{attribute 'hide' := ''}
	_rStopCmdTrig: R_TRIG;
	///当前运行的次数
	{attribute 'hide' := ''}
	_iActRunNumber: INT;
	{attribute 'hide' := ''}
	_wFluVolumeSetTemp: WORD;
	{attribute 'hide' := ''}
	_wRuntimeSetTemp: WORD;
	{attribute 'hide' := ''}
	_wSpeedSetTemp: WORD;
	{attribute 'hide' := ''}
	_rSetSpeed: REAL;
	{attribute 'hide' := ''}
	_wModuleSpeedSetTemp: WORD;
	{attribute 'hide' := ''}
	_wModuleRealVolumeTemp: WORD;
	{attribute 'hide' := ''}
	_rHMIControl: R_TRIG;
	{attribute 'hide' := ''}
	dwTest1: DWORD;
	///NG 计数
	{attribute 'hide' := ''}
	_iNGCount: INT;
	{attribute 'hide' := ''}
	_rOperaTrig: ARRAY[1..15] OF R_TRIG;
	{attribute 'hide' := ''}
	k: INT;
	{attribute 'hide' := ''}
	_bChannelNum: BYTE;
	_bDiagData: BYTE;
	{attribute 'hide' := ''}
	xAutomodeFlag: BOOL;
	{attribute 'hide' := ''}
	diStepOld: DINT;
	{attribute 'hide' := ''}
	st_IOData: RudongPump_IOData_1;
	{attribute 'hide' := ''}
	iPumpType: INT;
	///是否有手动操作，是否有自动操作	
	{attribute 'hide' := ''}
	_xHMIOpe: BOOL;
	///是否有手动操作，是否有自动操作	
	{attribute 'hide' := ''}
	_xAutoOpe: BOOL;
	{attribute 'hide' := ''}
	_rInit: R_TRIG;
	{attribute 'hide' := ''}
	_first: BOOL;
END_VAR
VAR_TEMP
	{attribute 'hide' := ''}
	xAgain: BOOL;
END_VAR

xAgain:=0;
//ConnectAction();//触发通信连接功能连接
ACTMap();//IO Map
IF NOT _first THEN
	_first:=TRUE;
ELSE

//只有在运行的时候，才会检测是否有模式切换发生
IF eState <> STATE.DORMANT
THEN	
	IF _rManual.Q OR _fManual.Q
	THEN
		_xModeChange := TRUE;//通知系统有模式切换发生
	END_IF
ELSE
	_xModeChange := FALSE;//待机状态不触发模式切换
END_IF

//检测是否是初始化中，如果是的去切换模式
_rInit(CLK:= xIniting);
IF _rInit.Q
THEN
	eState := STATE.RESETING;
END_IF	

REPEAT
	CASE eState OF
		STATE.DORMANT:
				HandleDormantState(xAgain=> xAgain);
		STATE.EXECUTING:
				HandleExecutingState(xAgain=> xAgain);
		STATE.DONE:
				HandleDoneState(xAgain=> xAgain);
		STATE.INERROR:
				HandleErrorState(xAgain=> xAgain);
		STATE.ABORTING:
				HandleAbortingState(xAgain=> xAgain);
		STATE.ABORTED:
				HandleAbortedState(xAgain=> xAgain);
		STATE.RESETING:
				HandleResettingState(xAgain=> xAgain);
	END_CASE
UNTIL (xAgain=0)
END_REPEAT
END_IF


//判断是否处于当前流程的Done状态
xDone := _xDone AND xExecute;
//输出报错信息
CASE eERRORID OF 	
  RudongPump_ERROR.No_ERROR:
		sHmiError:='No_ERROR';	
  RudongPump_ERROR.FLT_PARA:
		sHmiError:='FLT_PARA';
  RudongPump_ERROR.FLT_CONNECT:
		sHmiError:='FLT_CONNECT';
  RudongPump_ERROR.FLT_RDYCMD:
		sHmiError:='FLT_RDYCMD';
	RudongPump_ERROR.FLT_CONFIGURE_PARA:
		sHmiError:='FLT_CONFIGURE_PARA';
	RudongPump_ERROR.FLT_FLUVOLUM_TIME_PARA:
		sHmiError:='FLT_FLUVOLUM_TIME_PARA';  
  RudongPump_ERROR.FLT_PUSH_TIMEOUT:
		sHmiError:='FLT_PUSH_TIMEOUT';
  RudongPump_ERROR.FLT_PULL_TIMEOUT:
		sHmiError:='FLT_PULL_TIMEOUT';
  RudongPump_ERROR.FLT_STOP_TIMEOUT:
		sHmiError:='FLT_STOP_TIMEOUT'; 
	RudongPump_ERROR.FLT_FULLSPEEDSTOP_TIMEOUT:
		sHmiError:='FLT_FULLSPEEDSTOP_TIMEOUT';
	RudongPump_ERROR.FLT_FULLSPEEDSTART_TIMEOUT:
		sHmiError:='FLT_FULLSPEEDSTART_TIMEOUT'; 
	RudongPump_ERROR.FLT_CMD_TIMEOUT:
		sHmiError:='FLT_CMD_TIMEOUT';
	RudongPump_ERROR.FLT_RUN_FALL:
		sHmiError:='FLT_RUN_FALL';
	RudongPump_ERROR.FLT_Mobdus:
		sHmiError:=_fbModbusTCP.sError;		
		
END_CASE
//手动自动操作检测
_xHMIOpe :=
			stDeviceOpe.xConfigure_Hmi OR 
			stDeviceOpe.xFullSpeedPull_Hmi OR 
			stDeviceOpe.xFullSpeedPush_Hmi OR 
			stDeviceOpe.xPull_Hmi[1] OR 
			stDeviceOpe.xPull_Hmi[2] OR 
			stDeviceOpe.xPull_Hmi[3] OR 
			stDeviceOpe.xPull_Hmi[4] OR 
			stDeviceOpe.xPull_Hmi[5] OR 			
			stDeviceOpe.xPumpCal_Hmi OR 
			stDeviceOpe.xPush_Hmi[1] OR 
			stDeviceOpe.xPush_Hmi[2] OR 
			stDeviceOpe.xPush_Hmi[3] OR 			
			stDeviceOpe.xPush_Hmi[4] OR 			
			stDeviceOpe.xPush_Hmi[5] OR 						
			stDeviceOpe.xResetCalcoeffCal_Hmi OR 
			stDeviceOpe.xStop_Hmi;
_xAutoOpe:=	
			stDeviceOpe.xConfigure_Auto OR 
            stDeviceOpe.xFullSpeedPull_Auto OR 
            stDeviceOpe.xFullSpeedPush_Auto OR 
            stDeviceOpe.xPull_Auto[1] OR 
            stDeviceOpe.xPull_Auto[2] OR 			
            stDeviceOpe.xPull_Auto[3] OR 			
            stDeviceOpe.xPull_Auto[4] OR 			
            stDeviceOpe.xPull_Auto[5] OR 			
            stDeviceOpe.xPumpCal_Auto OR 
            stDeviceOpe.xPush_Auto[1] OR 
            stDeviceOpe.xPush_Auto[2] OR 			
            stDeviceOpe.xPush_Auto[3] OR 			
            stDeviceOpe.xPush_Auto[4] OR 			
            stDeviceOpe.xPush_Auto[5] OR 						
            stDeviceOpe.xStop_Auto;

METHOD PROTECTED AbortAction
VAR_OUTPUT
	xComplete: BOOL;
	eERRORID: RudongPump_ERROR;
END_VAR
(*
* Cleaning
* => abort all running operation
* => if an NBS.RudongPump_ERROR codition is reached, set eERRORID to a Value rather then NBS.RudongPump_ERROR.No_ERROR 
*)
xComplete:=1;
eERRORID:=RudongPump_ERROR.No_ERROR;
END_METHOD

ACTION ACT_GetModbusAddress:
//
(*************************检测配置参数是否匹配成功*********************************)
IF stRunPara.iPumpType=RudongPump_PumpType.DFPluse THEN//DF600Plus/KF300系列
	stModbusAddress.iPumpType_Address:=1000;
	stModbusAddress.iHosePipeType_Address:=1001;	
	stModbusAddress.iFluVolumeSet_Address:=1002;
	stModbusAddress.iRuntimeSet_Address:=1004;
	stModbusAddress.iIntervalTime_Address:=1006;
	stModbusAddress.iCycleNumber_Address:=1008;
	stModbusAddress.iBackAngle_Address:=1009;
	stModbusAddress.iMoveDirection_Address:=1010;
	stModbusAddress.iStartStop_Address:=1011;
	stModbusAddress.iFullSpeedStartStop_Address:=1012;
	stModbusAddress.iModuleAddress_Address:=2000;
	stModbusAddress.iModuleStartStop_Address:=2003;
	stModbusAddress.iModuleRealFluVolumeSet_Address:=2004;
	stModbusAddress.iRecoveryCalCoefficient_Address:=2007;	

ELSIF stRunPara.iPumpType=RudongPump_PumpType.F OR 
			stRunPara.iPumpType=RudongPump_PumpType.LabF1 OR
			stRunPara.iPumpType=RudongPump_PumpType.LabF3 OR
			stRunPara.iPumpType=RudongPump_PumpType.LabF4
THEN
	stModbusAddress.iPumpType_Address:=1000;
	stModbusAddress.iHosePipeType_Address:=1001;	
	stModbusAddress.iFluVolumeSet_Address:=1015;
	stModbusAddress.iRuntimeSet_Address:=1018;
	stModbusAddress.iIntervalTime_Address:=1021;
	stModbusAddress.iCycleNumber_Address:=1023;
	stModbusAddress.iBackAngle_Address:=1007;
	stModbusAddress.iMoveDirection_Address:=1009;
	stModbusAddress.iStartStop_Address:=1008;
	stModbusAddress.iFullSpeedStartStop_Address:=1010;
	stModbusAddress.iModuleAddress_Address:=0;//等于0表示不写入
	stModbusAddress.iModuleStartStop_Address:=2003;
	stModbusAddress.iModuleRealFluVolumeSet_Address:=2004;
	stModbusAddress.iRecoveryCalCoefficient_Address:=2006;	

